RoboDK station: KR200-2_Roboforming_Escala_Laboratorio.rdk

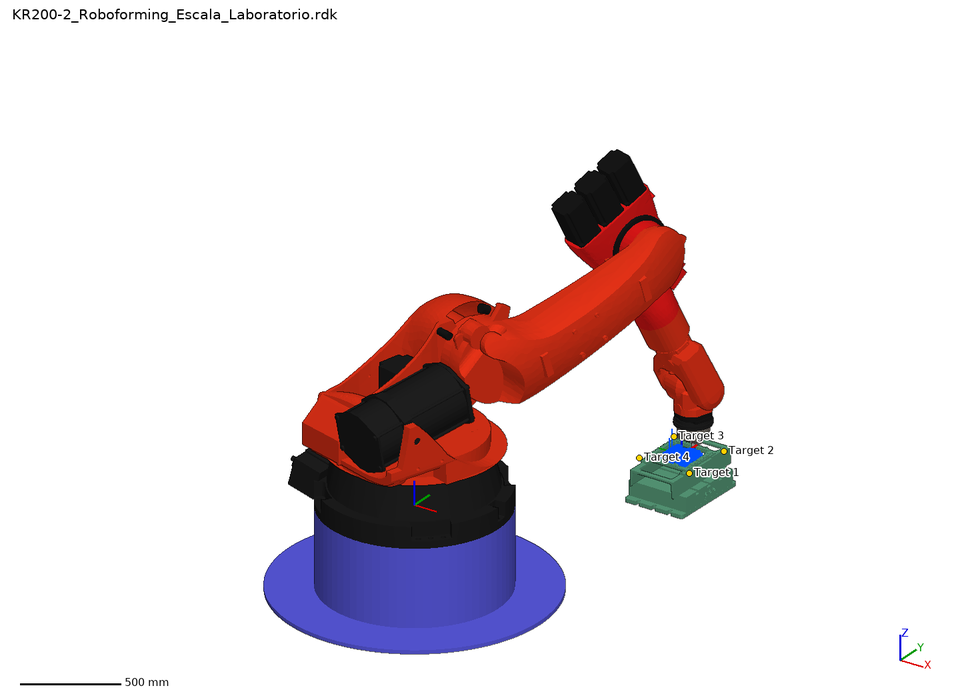
[picture v0: the station drawn from its stored meshes, robots at their saved joint values, targets as dots, program paths as lines]
Station KR200-2_Roboforming_Escala_Laboratorio (saved by RoboDK 5.8.0). Poses are relative to the parent item; angles as X-Y-Z fixed-axis rotations.
Station parameters (name, value as stored): IO_5, 1
  - frame KR200-2 comp Base at (0, 0, 458.56) mm
    - robot KR200-2 comp: 6 axes
        modified DH rows (alpha deg, a mm, theta deg, d mm): 0, 0, 0, 750; -90, 350, 0, 0; 0, 1050, -90, 0; -90, -45, 0, 1000; 90, 0, 0, 0; -90, 0, 180, 210
        joint limits [-185, -142, -120, -350, -120, -350] to [185, 0, 148, 350, 120, 350]; home [0, -90, 90, 0, 0, 0]; saved at [73.183, -16.623, 80.288, 0, 26.334, 73.183]
      - tool Kitagawa JN06T, TCP at (0, 0, 200) mm, size 164.9 x 165.3 x 101 mm, geometry from Kitagawa JN06T.STEP
      - tool herramienta_spif, TCP at (0, 0, 170) mm, size 17.5 x 18 x 175 mm, geometry from herramienta_spif.STEP
      - tool SPIF_TOOL, TCP at (0, 0, 170) mm, size 59.8 x 60 x 80 mm, geometry from SPIF_TOOL.stl
    - frame Machining at (474.42, 1634.58, -244.56) mm, rotated rx 0 ry 0 rz 90 deg
      - object myPart at (0, 0, 0) mm, size 300 x 300 x 40 mm, geometry from myPart.STP
        - object myToolpath_topToolTipPnts at (0, 0, 0) mm
      - target Target 1 (Cartesian target) at (-150, -150, 0) mm, rotated rx 179.98 ry -0.02 rz -135 deg; joints [14.532, -78.087, 109.692, 0.007, 58.419, -30.472] of KR200-2 comp
      - target Target 2 (Cartesian target) at (150, -150, 0) mm, rotated rx 179.98 ry -0.02 rz -135 deg; joints [11.975, -64.118, 90.175, 0.006, 63.968, -33.028] of KR200-2 comp
      - target Target 3 (Cartesian target) at (150, 150, 0) mm, rotated rx 179.98 ry -0.02 rz -135 deg; joints [21.499, -59.92, 83.648, 0.01, 66.295, -23.505] of KR200-2 comp
      - target Target 4 (Cartesian target) at (-150, 150, 0) mm, rotated rx 179.98 ry -0.02 rz -135 deg; joints [25.706, -73.09, 103.133, 0.013, 59.98, -19.3] of KR200-2 comp
  - machining project Machining1 settings: F:/SPIF.ptp | rotZ(0) | rotX(0)*rotY(0)
  - program Machining1 (10854 instructions, listed below)
  - object dispositivo sin pieza at (474.42, 1634.58, 214) mm, rotated rx 0 ry 0 rz 90 deg, size 500 x 358.5 x 227 mm, geometry from dispositivo sin pieza.STEP
  - object Base at (0, 0, 0) mm, size 1499.1 x 1499.1 x 458.6 mm, geometry from Base.IGS
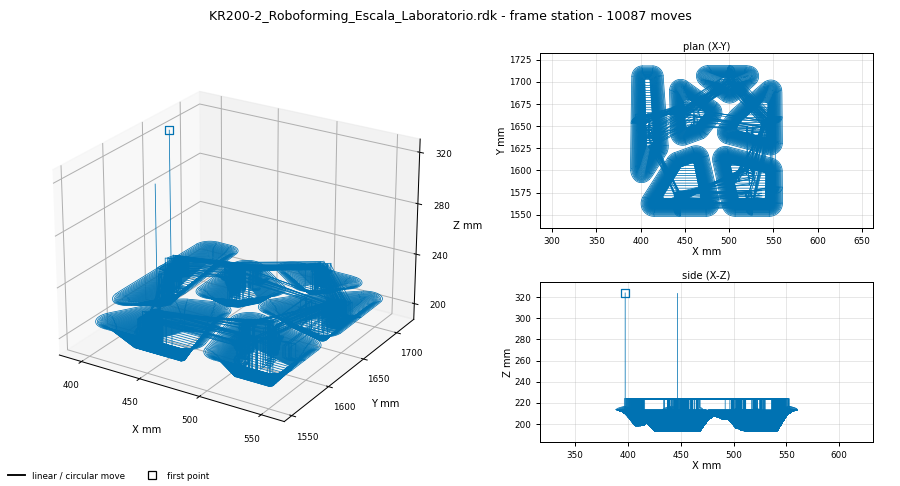
[picture p0: tool path of KR200-2_Roboforming_Escala_Laboratorio.rdk in frame station, 10087 of 10087 moves have a stored position in this frame; points joined in program order, loops and branches not executed]

--- program Machining1 (robot KR200-2 comp) ---
  Suave(1)
  Llamar SetTool(1)
  Llamar M_RunCode(6)
  Llamar SetRPM(0.0)
  Llamar M_RunCode(3)
  Establecer velocidad (1000.0 mm/s)
  Est. Ref.: Machining
  Est. herr: SPIF_TOOL
  Mostrar SPIF_TOOL
  MoveJ 1 to (25.11, 76.92, 110) mm, rotated rx 180 ry 0 rz 90 deg; joints [76.531, -23.354, 87.682, 0, 25.671, 76.531]
  MoveL 2 to (25.11, 76.92, 110) mm, rotated rx 180 ry 0 rz 90 deg; joints [76.531, -23.354, 87.682, 0, 25.671, 76.531]
  MoveL 3 to (25.11, 76.92, 10) mm, rotated rx -180 ry 0 rz 90 deg; joints [76.531, -18.294, 84.658, 0, 23.636, 76.531]
  MoveL 4 to (25.11, 76.92, 10) mm, rotated rx -180 ry 0 rz 90 deg; joints [76.531, -18.294, 84.658, 0, 23.636, 76.531]
  MoveL 5 to (25.11, 76.92, 10) mm, rotated rx -180 ry 0 rz 90 deg; joints [76.531, -18.294, 84.658, 0, 23.636, 76.531]
  MoveL 6 to (25.11, 76.92, 3) mm, rotated rx 180 ry 0 rz 90 deg; joints [76.531, -17.937, 84.426, 0, 23.511, 76.531]
  Establecer velocidad (66.7 mm/s)
  MoveL 7 to (25.32, 78.42, 2.59) mm, rotated rx 180 ry 0 rz 90 deg; joints [76.582, -17.919, 84.424, 0, 23.496, 76.582]
  MoveL 8 to (25.15, 79.93, 2.19) mm, rotated rx -180 ry 0 rz 90 deg; joints [76.63, -17.909, 84.448, 0, 23.461, 76.63]
  MoveL 9 to (24.66, 81.37, 1.78) mm, rotated rx -180 ry 0 rz 90 deg; joints [76.673, -17.904, 84.494, 0, 23.409, 76.673]
  MoveL 10 to (23.86, 82.66, 1.37) mm, rotated rx 180 ry 0 rz 90 deg; joints [76.709, -17.904, 84.56, 0, 23.344, 76.709]
  MoveL 11 to (22.79, 83.75, 0.97) mm, rotated rx 180 ry 0 rz 90 deg; joints [76.736, -17.908, 84.641, 0, 23.266, 76.736]
  MoveL 12 to (21.51, 84.57, 0.56) mm, rotated rx -180 ry 0 rz 90 deg; joints [76.753, -17.915, 84.734, 0, 23.181, 76.753]
  MoveL 13 to (20.09, 85.08, 0.16) mm, rotated rx 180 ry 0 rz 90 deg; joints [76.759, -17.923, 84.831, 0, 23.092, 76.759]
  MoveL 14 to (18.58, 85.24, -0.25) mm, rotated rx -180 ry 0 rz 90 deg; joints [76.753, -17.931, 84.928, 0, 23.002, 76.753]
  MoveL 15 to (-29.85, 85.86, -0.25) mm, rotated rx -180 ry 0 rz 90 deg; joints [76.389, -18.776, 88.341, 0, 20.435, 76.389]
  MoveL 16 to (-34.65, 85.65, -0.25) mm, rotated rx -180 ry 0 rz 90 deg; joints [76.342, -18.853, 88.668, 0, 20.185, 76.342]
  MoveC 17 to (-41.94, 83.49, -0.25) mm, rotated rx -180 ry 0 rz 90 deg; joints [76.209, -18.961, 89.132, 0, 19.829, 76.209] to (-47.38, 78.18, -0.25) mm, rotated rx -180 ry 0 rz 90 deg; joints [75.983, -19.025, 89.413, 0, 19.612, 75.983]
  MoveC 18 to (-48.12, 71.04, -0.25) mm, rotated rx 180 ry 0 rz 90 deg; joints [75.734, -19.009, 89.34, 0, 19.668, 75.734] to (-44.7, 64.73, -0.25) mm, rotated rx 180 ry 0 rz 90 deg; joints [75.55, -18.93, 88.997, 0, 19.932, 75.55]
  MoveL 19 to (-43.12, 63.19, -0.25) mm, rotated rx 180 ry 0 rz 90 deg; joints [75.512, -18.898, 88.862, 0, 20.036, 75.512]
  MoveL 20 to (-40.5, 61.12, -0.25) mm, rotated rx 180 ry 0 rz 90 deg; joints [75.465, -18.848, 88.647, 0, 20.201, 75.465]
  MoveL 21 to (-15.64, 45.37, -0.25) mm, rotated rx 180 ry 0 rz 90 deg; joints [75.157, -18.366, 86.643, 0, 21.723, 75.157]
  MoveL 22 to (-14.69, 44.91, -0.25) mm, rotated rx -180 ry 0 rz 90 deg; joints [75.15, -18.347, 86.568, 0, 21.779, 75.15]
  MoveC 23 to (-10.63, 43.57, -0.25) mm, rotated rx -180 ry 0 rz 90 deg; joints [75.141, -18.27, 86.259, 0, 22.011, 75.141] to (-6.36, 43.32, -0.25) mm, rotated rx 180 ry 0 rz 90 deg; joints [75.17, -18.193, 85.955, 0, 22.239, 75.17]
  MoveL 24 to (58.28, 48.02, -0.25) mm, rotated rx -180 ry 0 rz 90 deg; joints [75.862, -16.971, 81.374, 0, 25.597, 75.862]
  MoveL 25 to (72.44, 48.99, -0.25) mm, rotated rx -180 ry 0 rz 90 deg; joints [76.006, -16.677, 80.335, 0, 26.342, 76.006]
  MoveC 26 to (80.2, 52.59, -0.25) mm, rotated rx -180 ry 0 rz 90 deg; joints [76.18, -16.528, 79.817, 0, 26.711, 76.18] to (83.56, 60.47, -0.25) mm, rotated rx 180 ry 0 rz 90 deg; joints [76.454, -16.496, 79.708, 0, 26.788, 76.454]
  MoveL 27 to (83.58, 61.12, -0.25) mm, rotated rx -180 ry 0 rz 90 deg; joints [76.475, -16.499, 79.718, 0, 26.781, 76.475]
  MoveL 28 to (83.58, 72.42, -0.25) mm, rotated rx 180 ry 0 rz 90 deg; joints [76.831, -16.558, 79.921, 0, 26.637, 76.831]
  MoveC 29 to (80.15, 80.83, -0.25) mm, rotated rx 180 ry 0 rz 90 deg; joints [77.073, -16.675, 80.328, 0, 26.347, 77.073] to (71.81, 84.44, -0.25) mm, rotated rx 180 ry 0 rz 90 deg; joints [77.127, -16.871, 81.017, 0, 25.854, 77.127]
  MoveL 30 to (54.49, 84.79, -0.25) mm, rotated rx -180 ry 0 rz 90 deg; joints [77.01, -17.231, 82.31, 0, 24.921, 77.01]
  MoveL 31 to (18.58, 85.24, -0.25) mm, rotated rx -180 ry 0 rz 90 deg; joints [76.753, -17.931, 84.928, 0, 23.002, 76.753]
  MoveL 32 to (18.48, 77.69, -0.25) mm, rotated rx -180 ry 0 rz 90 deg; joints [76.505, -17.899, 84.807, 0, 23.093, 76.505]
  MoveL 33 to (18.48, 77.69, 2.75) mm, rotated rx -180 ry 0 rz 90 deg; joints [76.505, -18.053, 84.907, 0, 23.146, 76.505]
  Establecer velocidad (1000.0 mm/s)
  MoveL 34 to (18.48, 77.69, 10) mm, rotated rx 180 ry 0 rz 90 deg; joints [76.505, -18.423, 85.148, 0, 23.276, 76.505]
  Establecer velocidad (66.7 mm/s)
  MoveL 35 to (38.08, 33.07, 10) mm, rotated rx 180 ry 0 rz 90 deg; joints [75.219, -17.824, 82.918, 0, 24.906, 75.219]
  MoveL 36 to (38.08, 33.07, 3) mm, rotated rx -180 ry 0 rz 90 deg; joints [75.219, -17.469, 82.685, 0, 24.784, 75.219]
  MoveL 37 to (38.23, 34.58, 2.59) mm, rotated rx 180 ry 0 rz 90 deg; joints [75.269, -17.454, 82.69, 0, 24.763, 75.269]
  MoveL 38 to (38, 36.09, 2.19) mm, rotated rx 180 ry 0 rz 90 deg; joints [75.315, -17.445, 82.722, 0, 24.723, 75.315]
  MoveL 39 to (37.45, 37.5, 1.78) mm, rotated rx -180 ry 0 rz 90 deg; joints [75.356, -17.443, 82.776, 0, 24.668, 75.356]
  MoveL 40 to (36.6, 38.76, 1.37) mm, rotated rx 180 ry 0 rz 90 deg; joints [75.389, -17.446, 82.848, 0, 24.598, 75.389]
  MoveL 41 to (35.49, 39.8, 0.97) mm, rotated rx 180 ry 0 rz 90 deg; joints [75.413, -17.453, 82.935, 0, 24.518, 75.413]
  MoveL 42 to (34.18, 40.57, 0.56) mm, rotated rx -180 ry 0 rz 90 deg; joints [75.427, -17.462, 83.031, 0, 24.431, 75.427]
  MoveL 43 to (32.74, 41.03, 0.16) mm, rotated rx -180 ry 0 rz 90 deg; joints [75.429, -17.472, 83.131, 0, 24.341, 75.429]
  MoveL 44 to (31.22, 41.13, -0.25) mm, rotated rx -180 ry 0 rz 90 deg; joints [75.42, -17.482, 83.229, 0, 24.252, 75.42]
  MoveL 45 to (7.11, 40.47, -0.25) mm, rotated rx -180 ry 0 rz 90 deg; joints [75.193, -17.936, 84.949, 0, 22.987, 75.193]
  MoveL 46 to (5.6, 40.3, -0.25) mm, rotated rx 180 ry 0 rz 90 deg; joints [75.175, -17.963, 85.052, 0, 22.911, 75.175]
  MoveC 47 to (-4.04, 34.34, -0.25) mm, rotated rx 180 ry 0 rz 90 deg; joints [74.896, -18.109, 85.622, 0, 22.487, 74.896] to (-5.53, 23.11, -0.25) mm, rotated rx -180 ry 0 rz 90 deg; joints [74.515, -18.081, 85.511, 0, 22.57, 74.515]
  MoveL 48 to (-4.96, 21.32, -0.25) mm, rotated rx -180 ry 0 rz 90 deg; joints [74.462, -18.062, 85.436, 0, 22.626, 74.462]
  MoveL 49 to (0.91, 5.21, -0.25) mm, rotated rx -180 ry 0 rz 90 deg; joints [73.992, -17.871, 84.699, 0, 23.172, 73.992]
  MoveL 50 to (1.74, 3.32, -0.25) mm, rotated rx 180 ry 0 rz 90 deg; joints [73.939, -17.846, 84.602, 0, 23.244, 73.939]
  MoveC 51 to (3.62, 0.75, -0.25) mm, rotated rx 180 ry 0 rz 90 deg; joints [73.873, -17.797, 84.416, 0, 23.382, 73.873] to (5.93, -1.42, -0.25) mm, rotated rx 180 ry 0 rz 90 deg; joints [73.825, -17.742, 84.206, 0, 23.536, 73.825]
  MoveL 52 to (22.27, -14.11, -0.25) mm, rotated rx -180 ry 0 rz 90 deg; joints [73.572, -17.357, 82.768, 0, 24.589, 73.572]
  MoveL 53 to (23.38, -14.89, -0.25) mm, rotated rx 180 ry 0 rz 90 deg; joints [73.557, -17.33, 82.671, 0, 24.659, 73.557]
  MoveC 54 to (33.35, -17.16, -0.25) mm, rotated rx -180 ry 0 rz 90 deg; joints [73.579, -17.117, 81.898, 0, 25.219, 73.579] to (42.02, -11.74, -0.25) mm, rotated rx -180 ry 0 rz 90 deg; joints [73.83, -16.973, 81.379, 0, 25.593, 73.83]
  MoveL 55 to (65.02, 20.37, -0.25) mm, rotated rx 180 ry 0 rz 90 deg; joints [75.043, -16.677, 80.337, 0, 26.34, 75.043]
  MoveL 56 to (66.39, 22.51, -0.25) mm, rotated rx 180 ry 0 rz 90 deg; joints [75.122, -16.66, 80.277, 0, 26.383, 75.122]
  MoveC 57 to (67.04, 34.78, -0.25) mm, rotated rx 180 ry 0 rz 90 deg; joints [75.514, -16.715, 80.469, 0, 26.246, 75.514] to (56.85, 41.63, -0.25) mm, rotated rx 180 ry 0 rz 90 deg; joints [75.648, -16.967, 81.36, 0, 25.607, 75.648]
  MoveL 58 to (55.44, 41.74, -0.25) mm, rotated rx 180 ry 0 rz 90 deg; joints [75.639, -16.997, 81.466, 0, 25.531, 75.639]
  MoveL 59 to (54.49, 41.77, -0.25) mm, rotated rx -180 ry 0 rz 90 deg; joints [75.633, -17.017, 81.537, 0, 25.48, 75.633]
  MoveL 60 to (31.22, 41.13, -0.25) mm, rotated rx -180 ry 0 rz 90 deg; joints [75.42, -17.482, 83.229, 0, 24.252, 75.42]
  MoveL 61 to (31.43, 33.58, -0.25) mm, rotated rx -180 ry 0 rz 90 deg; joints [75.179, -17.439, 83.071, 0, 24.368, 75.179]
  MoveL 62 to (31.43, 33.58, 2.75) mm, rotated rx -180 ry 0 rz 90 deg; joints [75.179, -17.591, 83.171, 0, 24.42, 75.179]
  Establecer velocidad (1000.0 mm/s)
  MoveL 63 to (31.43, 33.58, 10) mm, rotated rx 180 ry 0 rz 90 deg; joints [75.179, -17.959, 83.412, 0, 24.547, 75.179]
  Establecer velocidad (66.7 mm/s)
  MoveL 64 to (75.76, -31.94, 10) mm, rotated rx 180 ry 0 rz 90 deg; joints [73.508, -16.63, 78.763, 0, 27.867, 73.508]
  MoveL 65 to (75.76, -31.94, 3) mm, rotated rx -180 ry 0 rz 90 deg; joints [73.508, -16.281, 78.529, 0, 27.752, 73.508]
  MoveL 66 to (77.26, -32.13, 2.59) mm, rotated rx 180 ry 0 rz 90 deg; joints [73.516, -16.225, 78.396, 0, 27.829, 73.516]
  MoveL 67 to (78.77, -31.95, 2.19) mm, rotated rx 180 ry 0 rz 90 deg; joints [73.535, -16.172, 78.272, 0, 27.9, 73.535]
  MoveL 68 to (80.2, -31.43, 1.78) mm, rotated rx 180 ry 0 rz 90 deg; joints [73.564, -16.123, 78.161, 0, 27.962, 73.564]
  MoveL 69 to (81.48, -30.62, 1.37) mm, rotated rx -180 ry 0 rz 90 deg; joints [73.601, -16.079, 78.068, 0, 28.011, 73.601]
  MoveL 70 to (82.56, -29.54, 0.97) mm, rotated rx 180 ry 0 rz 90 deg; joints [73.644, -16.041, 77.997, 0, 28.045, 73.644]
  MoveL 71 to (83.36, -28.25, 0.56) mm, rotated rx -180 ry 0 rz 90 deg; joints [73.69, -16.011, 77.95, 0, 28.061, 73.69]
  MoveL 72 to (83.86, -26.81, 0.16) mm, rotated rx -180 ry 0 rz 90 deg; joints [73.739, -15.989, 77.93, 0, 28.059, 73.739]
  MoveL 73 to (84, -25.3, -0.25) mm, rotated rx -180 ry 0 rz 90 deg; joints [73.787, -15.976, 77.94, 0, 28.036, 73.787]
  MoveL 74 to (84, -4.26, -0.25) mm, rotated rx -180 ry 0 rz 90 deg; joints [74.436, -16.112, 78.397, 0, 27.715, 74.436]
  MoveL 75 to (83.9, -1.36, -0.25) mm, rotated rx 180 ry 0 rz 90 deg; joints [74.525, -16.132, 78.466, 0, 27.667, 74.525]
  MoveC 76 to (81.73, 5.7, -0.25) mm, rotated rx -180 ry 0 rz 90 deg; joints [74.725, -16.225, 78.779, 0, 27.446, 74.725] to (76.29, 10.7, -0.25) mm, rotated rx -180 ry 0 rz 90 deg; joints [74.835, -16.376, 79.294, 0, 27.082, 74.835]
  MoveC 77 to (69.05, 10.89, -0.25) mm, rotated rx 180 ry 0 rz 90 deg; joints [74.779, -16.535, 79.844, 0, 26.692, 74.779] to (62.94, 7.01, -0.25) mm, rotated rx -180 ry 0 rz 90 deg; joints [74.605, -16.644, 80.222, 0, 26.423, 74.605]
  MoveL 78 to (60.58, 4.26, -0.25) mm, rotated rx 180 ry 0 rz 90 deg; joints [74.499, -16.679, 80.341, 0, 26.337, 74.499]
  MoveL 79 to (44.7, -17.53, -0.25) mm, rotated rx -180 ry 0 rz 90 deg; joints [73.672, -16.882, 81.058, 0, 25.824, 73.672]
  MoveL 80 to (43.76, -18.94, -0.25) mm, rotated rx 180 ry 0 rz 90 deg; joints [73.619, -16.893, 81.097, 0, 25.797, 73.619]
  MoveC 81 to (41.63, -26.99, -0.25) mm, rotated rx 180 ry 0 rz 90 deg; joints [73.346, -16.888, 81.078, 0, 25.81, 73.346] to (44.86, -34.66, -0.25) mm, rotated rx -180 ry 0 rz 90 deg; joints [73.137, -16.772, 80.669, 0, 26.103, 73.137]
  MoveL 82 to (62.52, -54.49, -0.25) mm, rotated rx -180 ry 0 rz 90 deg; joints [72.69, -16.261, 78.901, 0, 27.36, 72.69]
  MoveL 83 to (63.6, -55.44, -0.25) mm, rotated rx -180 ry 0 rz 90 deg; joints [72.671, -16.23, 78.797, 0, 27.433, 72.671]
  MoveL 84 to (64.56, -56.24, -0.25) mm, rotated rx -180 ry 0 rz 90 deg; joints [72.656, -16.204, 78.707, 0, 27.497, 72.656]
  MoveC 85 to (75.98, -58.19, -0.25) mm, rotated rx -180 ry 0 rz 90 deg; joints [72.705, -15.933, 77.796, 0, 28.137, 72.705] to (83.3, -49.2, -0.25) mm, rotated rx 180 ry 0 rz 90 deg; joints [73.048, -15.829, 77.449, 0, 28.38, 73.048]
  MoveL 86 to (83.95, -45.01, -0.25) mm, rotated rx -180 ry 0 rz 90 deg; joints [73.182, -15.843, 77.496, 0, 28.346, 73.182]
  MoveL 87 to (84, -44.07, -0.25) mm, rotated rx -180 ry 0 rz 90 deg; joints [73.212, -15.848, 77.515, 0, 28.334, 73.212]
  MoveL 88 to (84, -25.3, -0.25) mm, rotated rx -180 ry 0 rz 90 deg; joints [73.787, -15.976, 77.94, 0, 28.036, 73.787]
  MoveL 89 to (76.45, -25.3, -0.25) mm, rotated rx 180 ry 0 rz 90 deg; joints [73.719, -16.147, 78.514, 0, 27.632, 73.719]
  MoveL 90 to (76.45, -25.3, 2.75) mm, rotated rx 180 ry 0 rz 90 deg; joints [73.719, -16.297, 78.616, 0, 27.681, 73.719]
  Establecer velocidad (1000.0 mm/s)
  MoveL 91 to (76.45, -25.3, 10) mm, rotated rx -180 ry 0 rz 90 deg; joints [73.719, -16.659, 78.859, 0, 27.8, 73.719]
  Establecer velocidad (66.7 mm/s)
  MoveL 92 to (19.29, -77.28, 10) mm, rotated rx -180 ry 0 rz 90 deg; joints [71.552, -17.537, 81.89, 0, 25.648, 71.552]
  MoveL 93 to (19.29, -77.28, 3) mm, rotated rx 180 ry 0 rz 90 deg; joints [71.552, -17.184, 81.656, 0, 25.527, 71.552]
  MoveL 94 to (19.12, -78.79, 2.59) mm, rotated rx 180 ry 0 rz 90 deg; joints [71.503, -17.157, 81.619, 0, 25.538, 71.503]
  MoveL 95 to (19.32, -80.3, 2.19) mm, rotated rx 180 ry 0 rz 90 deg; joints [71.458, -17.122, 81.554, 0, 25.568, 71.458]
  MoveL 96 to (19.85, -81.72, 1.78) mm, rotated rx 180 ry 0 rz 90 deg; joints [71.42, -17.081, 81.468, 0, 25.613, 71.42]
  MoveL 97 to (20.67, -83, 1.37) mm, rotated rx 180 ry 0 rz 90 deg; joints [71.389, -17.035, 81.363, 0, 25.672, 71.389]
  MoveL 98 to (21.76, -84.06, 0.97) mm, rotated rx 180 ry 0 rz 90 deg; joints [71.367, -16.985, 81.244, 0, 25.74, 71.367]
  MoveL 99 to (23.06, -84.85, 0.56) mm, rotated rx 180 ry 0 rz 90 deg; joints [71.356, -16.932, 81.117, 0, 25.815, 71.356]
  MoveL 100 to (24.5, -85.34, 0.16) mm, rotated rx 180 ry 0 rz 90 deg; joints [71.356, -16.879, 80.987, 0, 25.892, 71.356]
  MoveL 101 to (26.01, -85.46, -0.25) mm, rotated rx -180 ry 0 rz 90 deg; joints [71.368, -16.826, 80.86, 0, 25.966, 71.368]
  MoveL 102 to (53.54, -85.2, -0.25) mm, rotated rx 180 ry 0 rz 90 deg; joints [71.659, -16.241, 78.834, 0, 27.407, 71.659]
  MoveL 103 to (56.28, -84.98, -0.25) mm, rotated rx -180 ry 0 rz 90 deg; joints [71.694, -16.182, 78.634, 0, 27.548, 71.694]
  MoveC 104 to (66.45, -77.93, -0.25) mm, rotated rx 180 ry 0 rz 90 deg; joints [72.011, -16.007, 78.043, 0, 27.964, 72.011] to (65.33, -65.6, -0.25) mm, rotated rx 180 ry 0 rz 90 deg; joints [72.376, -16.121, 78.426, 0, 27.694, 72.376]
  MoveL 105 to (63.5, -63.02, -0.25) mm, rotated rx 180 ry 0 rz 90 deg; joints [72.438, -16.18, 78.626, 0, 27.554, 72.438]
  MoveL 106 to (34.59, -29.56, -0.25) mm, rotated rx 180 ry 0 rz 90 deg; joints [73.199, -17.017, 81.538, 0, 25.48, 73.199]
  MoveL 107 to (33.64, -28.5, -0.25) mm, rotated rx 180 ry 0 rz 90 deg; joints [73.223, -17.043, 81.63, 0, 25.413, 73.223]
  MoveL 108 to (33.08, -27.96, -0.25) mm, rotated rx -180 ry 0 rz 90 deg; joints [73.235, -17.058, 81.683, 0, 25.374, 73.235]
  MoveL 109 to (17.53, -15.48, -0.25) mm, rotated rx 180 ry 0 rz 90 deg; joints [73.483, -17.441, 83.081, 0, 24.361, 73.483]
  MoveL 110 to (15.92, -14.42, -0.25) mm, rotated rx 180 ry 0 rz 90 deg; joints [73.502, -17.479, 83.219, 0, 24.26, 73.502]
  MoveC 111 to (3.85, -13.12, -0.25) mm, rotated rx 180 ry 0 rz 90 deg; joints [73.429, -17.717, 84.109, 0, 23.607, 73.429] to (-4.25, -22.15, -0.25) mm, rotated rx -180 ry 0 rz 90 deg; joints [73.06, -17.817, 84.492, 0, 23.326, 73.06]
  MoveL 112 to (-16.58, -68.7, -0.25) mm, rotated rx 180 ry 0 rz 90 deg; joints [71.444, -17.769, 84.31, 0, 23.46, 71.444]
  MoveC 113 to (-14.48, -80.13, -0.25) mm, rotated rx -180 ry 0 rz 90 deg; joints [71.104, -17.659, 83.89, 0, 23.768, 71.104] to (-4.26, -85.66, -0.25) mm, rotated rx -180 ry 0 rz 90 deg; joints [71.04, -17.429, 83.034, 0, 24.395, 71.04]
  MoveL 114 to (-2.37, -85.73, -0.25) mm, rotated rx -180 ry 0 rz 90 deg; joints [71.059, -17.392, 82.897, 0, 24.494, 71.059]
  MoveL 115 to (26.01, -85.46, -0.25) mm, rotated rx -180 ry 0 rz 90 deg; joints [71.368, -16.826, 80.86, 0, 25.966, 71.368]
  MoveL 116 to (25.94, -77.91, -0.25) mm, rotated rx -180 ry 0 rz 90 deg; joints [71.602, -16.88, 81.049, 0, 25.831, 71.602]
  MoveL 117 to (25.94, -77.91, 2.75) mm, rotated rx -180 ry 0 rz 90 deg; joints [71.602, -17.031, 81.15, 0, 25.881, 71.602]
  Establecer velocidad (1000.0 mm/s)
  MoveL 118 to (25.94, -77.91, 10) mm, rotated rx 180 ry 0 rz 90 deg; joints [71.602, -17.396, 81.392, 0, 26.004, 71.602]
  Establecer velocidad (66.7 mm/s)
  MoveL 119 to (-60.09, -77.51, 10) mm, rotated rx -180 ry 0 rz 90 deg; joints [70.682, -19.008, 87.445, 0, 21.563, 70.682]
  MoveL 120 to (-60.09, -77.51, 3) mm, rotated rx 180 ry 0 rz 90 deg; joints [70.682, -18.647, 87.213, 0, 21.434, 70.682]
  MoveL 121 to (-60.27, -79.01, 2.59) mm, rotated rx 180 ry 0 rz 90 deg; joints [70.631, -18.62, 87.175, 0, 21.445, 70.631]
  MoveL 122 to (-60.07, -80.52, 2.19) mm, rotated rx -180 ry 0 rz 90 deg; joints [70.585, -18.587, 87.113, 0, 21.474, 70.585]
  MoveL 123 to (-59.55, -81.95, 1.78) mm, rotated rx -180 ry 0 rz 90 deg; joints [70.545, -18.549, 87.029, 0, 21.52, 70.545]
  MoveL 124 to (-58.72, -83.22, 1.37) mm, rotated rx -180 ry 0 rz 90 deg; joints [70.513, -18.507, 86.929, 0, 21.577, 70.513]
  MoveL 125 to (-57.64, -84.28, 0.97) mm, rotated rx -180 ry 0 rz 90 deg; joints [70.491, -18.461, 86.816, 0, 21.645, 70.491]
  MoveL 126 to (-56.34, -85.08, 0.56) mm, rotated rx 180 ry 0 rz 90 deg; joints [70.48, -18.414, 86.695, 0, 21.718, 70.48]
  MoveL 127 to (-54.9, -85.57, 0.16) mm, rotated rx 180 ry 0 rz 90 deg; joints [70.481, -18.366, 86.572, 0, 21.794, 70.481]
  MoveL 128 to (-53.39, -85.69, -0.25) mm, rotated rx -180 ry 0 rz 90 deg; joints [70.494, -18.318, 86.452, 0, 21.866, 70.494]
  MoveL 129 to (-35.3, -85.56, -0.25) mm, rotated rx -180 ry 0 rz 90 deg; joints [70.703, -18.004, 85.212, 0, 22.792, 70.703]
  MoveC 130 to (-26.15, -82.38, -0.25) mm, rotated rx 180 ry 0 rz 90 deg; joints [70.905, -17.859, 84.654, 0, 23.206, 70.905] to (-20.83, -74.28, -0.25) mm, rotated rx -180 ry 0 rz 90 deg; joints [71.221, -17.813, 84.476, 0, 23.337, 71.221]
  MoveL 131 to (-8.05, -25.1, -0.25) mm, rotated rx -180 ry 0 rz 90 deg; joints [72.928, -17.871, 84.696, 0, 23.174, 72.928]
  MoveC 132 to (-11.52, -11.33, -0.25) mm, rotated rx -180 ry 0 rz 90 deg; joints [73.339, -18.01, 85.234, 0, 22.776, 73.339] to (-25.11, -7.26, -0.25) mm, rotated rx -180 ry 0 rz 90 deg; joints [73.339, -18.272, 86.269, 0, 22.004, 73.339]
  MoveL 133 to (-74.68, -17.81, -0.25) mm, rotated rx 180 ry 0 rz 90 deg; joints [72.487, -19.028, 89.426, 0, 19.602, 72.487]
  MoveC 134 to (-83.14, -22.99, -0.25) mm, rotated rx 180 ry 0 rz 90 deg; joints [72.223, -19.131, 89.88, 0, 19.25, 72.223] to (-86.46, -32.35, -0.25) mm, rotated rx 180 ry 0 rz 90 deg; joints [71.874, -19.135, 89.899, 0, 19.236, 71.874]
  MoveL 135 to (-86.48, -70.94, -0.25) mm, rotated rx -180 ry 0 rz 90 deg; joints [70.594, -18.937, 89.03, 0, 19.907, 70.594]
  MoveC 136 to (-82.08, -81.51, -0.25) mm, rotated rx 180 ry 0 rz 90 deg; joints [70.298, -18.811, 88.488, 0, 20.323, 70.298] to (-71.48, -85.83, -0.25) mm, rotated rx -180 ry 0 rz 90 deg; joints [70.281, -18.618, 87.674, 0, 20.943, 70.281]
  MoveL 137 to (-53.39, -85.69, -0.25) mm, rotated rx -180 ry 0 rz 90 deg; joints [70.494, -18.318, 86.452, 0, 21.866, 70.494]
  MoveL 138 to (-53.45, -78.15, -0.25) mm, rotated rx 180 ry 0 rz 90 deg; joints [70.737, -18.364, 86.637, 0, 21.727, 70.737]
  MoveL 139 to (-53.45, -78.15, 2.75) mm, rotated rx 180 ry 0 rz 90 deg; joints [70.737, -18.519, 86.738, 0, 21.781, 70.737]
  Establecer velocidad (1000.0 mm/s)
  MoveL 140 to (-53.45, -78.15, 10) mm, rotated rx -180 ry 0 rz 90 deg; joints [70.737, -18.892, 86.978, 0, 21.914, 70.737]
  Establecer velocidad (66.7 mm/s)
  MoveL 141 to (-78.23, 36.45, 10) mm, rotated rx 180 ry 0 rz 90 deg; joints [74.283, -19.86, 91.085, 0, 18.775, 74.283]
  MoveL 142 to (-78.23, 36.45, 3) mm, rotated rx -180 ry 0 rz 90 deg; joints [74.283, -19.493, 90.853, 0, 18.64, 74.283]
  MoveL 143 to (-79.74, 36.64, 2.59) mm, rotated rx -180 ry 0 rz 90 deg; joints [74.275, -19.494, 90.943, 0, 18.551, 74.275]
  MoveL 144 to (-81.24, 36.45, 2.19) mm, rotated rx 180 ry 0 rz 90 deg; joints [74.254, -19.493, 91.026, 0, 18.468, 74.254]
  MoveL 145 to (-82.67, 35.94, 1.78) mm, rotated rx -180 ry 0 rz 90 deg; joints [74.223, -19.491, 91.098, 0, 18.393, 74.223]
  MoveL 146 to (-83.96, 35.13, 1.37) mm, rotated rx 180 ry 0 rz 90 deg; joints [74.182, -19.484, 91.154, 0, 18.33, 74.182]
  MoveL 147 to (-85.03, 34.05, 0.97) mm, rotated rx -180 ry 0 rz 90 deg; joints [74.135, -19.474, 91.191, 0, 18.283, 74.135]
  MoveL 148 to (-85.83, 32.76, 0.56) mm, rotated rx 180 ry 0 rz 90 deg; joints [74.083, -19.459, 91.206, 0, 18.252, 74.083]
  MoveL 149 to (-86.33, 31.32, 0.16) mm, rotated rx -180 ry 0 rz 90 deg; joints [74.029, -19.439, 91.199, 0, 18.24, 74.029]
  MoveL 150 to (-86.47, 29.81, -0.25) mm, rotated rx 180 ry 0 rz 90 deg; joints [73.976, -19.413, 91.166, 0, 18.247, 73.976]
  MoveL 151 to (-86.47, 0.4, -0.25) mm, rotated rx -180 ry 0 rz 90 deg; joints [72.976, -19.288, 90.588, 0, 18.7, 72.976]
  MoveC 152 to (-80.93, -11.12, -0.25) mm, rotated rx -180 ry 0 rz 90 deg; joints [72.645, -19.154, 89.983, 0, 19.171, 72.645] to (-68.46, -13.96, -0.25) mm, rotated rx 180 ry 0 rz 90 deg; joints [72.68, -18.951, 89.09, 0, 19.861, 72.68]
  MoveL 153 to (-58.28, -11.64, -0.25) mm, rotated rx -180 ry 0 rz 90 deg; joints [72.863, -18.803, 88.452, 0, 20.35, 72.863]
  MoveL 154 to (-19.43, -2.7, -0.25) mm, rotated rx -180 ry 0 rz 90 deg; joints [73.543, -18.197, 85.967, 0, 22.229, 73.543]
  MoveL 155 to (-17.83, -2.31, -0.25) mm, rotated rx 180 ry 0 rz 90 deg; joints [73.571, -18.17, 85.864, 0, 22.307, 73.571]
  MoveC 156 to (-8.42, 4.98, -0.25) mm, rotated rx 180 ry 0 rz 90 deg; joints [73.898, -18.04, 85.353, 0, 22.687, 73.898] to (-7.54, 16.85, -0.25) mm, rotated rx 180 ry 0 rz 90 deg; joints [74.292, -18.085, 85.529, 0, 22.556, 74.292]
  MoveL 157 to (-14.62, 36.55, -0.25) mm, rotated rx 180 ry 0 rz 90 deg; joints [74.875, -18.307, 86.407, 0, 21.9, 74.875]
  MoveC 158 to (-17.05, 40.7, -0.25) mm, rotated rx -180 ry 0 rz 90 deg; joints [74.99, -18.368, 86.654, 0, 21.714, 74.99] to (-20.65, 43.89, -0.25) mm, rotated rx -180 ry 0 rz 90 deg; joints [75.064, -18.445, 86.964, 0, 21.481, 75.064]
  MoveL 159 to (-63.02, 71.07, -0.25) mm, rotated rx 180 ry 0 rz 90 deg; joints [75.605, -19.235, 90.349, 0, 18.886, 75.605]
  MoveL 160 to (-64.91, 72.11, -0.25) mm, rotated rx 180 ry 0 rz 90 deg; joints [75.624, -19.267, 90.494, 0, 18.773, 75.624]
  MoveC 161 to (-79.41, 71.9, -0.25) mm, rotated rx -180 ry 0 rz 90 deg; joints [75.489, -19.476, 91.46, 0, 18.016, 75.489] to (-86.47, 59.23, -0.25) mm, rotated rx 180 ry 0 rz 90 deg; joints [74.987, -19.528, 91.706, 0, 17.822, 74.987]
  MoveL 162 to (-86.47, 29.81, -0.25) mm, rotated rx 180 ry 0 rz 90 deg; joints [73.976, -19.413, 91.166, 0, 18.247, 73.976]
  MoveL 163 to (-78.92, 29.81, -0.25) mm, rotated rx 180 ry 0 rz 90 deg; joints [74.05, -19.305, 90.664, 0, 18.64, 74.05]
  MoveL 164 to (-78.92, 29.81, 2.75) mm, rotated rx 180 ry 0 rz 90 deg; joints [74.05, -19.462, 90.765, 0, 18.697, 74.05]
  Establecer velocidad (1000.0 mm/s)
  MoveL 165 to (-78.92, 29.81, 10) mm, rotated rx -180 ry 0 rz 90 deg; joints [74.05, -19.843, 91.006, 0, 18.837, 74.05]
  Establecer velocidad (66.7 mm/s)
  MoveL 166 to (-77, 36.45, 10) mm, rotated rx -180 ry 0 rz 90 deg; joints [74.295, -19.842, 91.003, 0, 18.839, 74.295]
  MoveL 167 to (-77, 36.45, 2.75) mm, rotated rx 180 ry 0 rz 90 deg; joints [74.295, -19.461, 90.762, 0, 18.699, 74.295]
  MoveL 168 to (-78.5, 36.64, 2.34) mm, rotated rx 180 ry 0 rz 90 deg; joints [74.287, -19.463, 90.852, 0, 18.611, 74.287]
  MoveL 169 to (-80.01, 36.45, 1.94) mm, rotated rx -180 ry 0 rz 90 deg; joints [74.266, -19.463, 90.936, 0, 18.527, 74.266]
  MoveL 170 to (-81.44, 35.94, 1.53) mm, rotated rx 180 ry 0 rz 90 deg; joints [74.235, -19.46, 91.007, 0, 18.452, 74.235]
  MoveL 171 to (-82.72, 35.13, 1.13) mm, rotated rx 180 ry 0 rz 90 deg; joints [74.194, -19.454, 91.064, 0, 18.39, 74.194]
  MoveL 172 to (-83.79, 34.05, 0.72) mm, rotated rx 180 ry 0 rz 90 deg; joints [74.147, -19.443, 91.101, 0, 18.342, 74.147]
  MoveL 173 to (-84.6, 32.76, 0.31) mm, rotated rx -180 ry 0 rz 90 deg; joints [74.095, -19.428, 91.116, 0, 18.312, 74.095]
  MoveL 174 to (-85.1, 31.32, -0.09) mm, rotated rx -180 ry 0 rz 90 deg; joints [74.041, -19.408, 91.108, 0, 18.299, 74.041]
  MoveL 175 to (-85.23, 29.81, -0.5) mm, rotated rx 180 ry 0 rz 90 deg; joints [73.988, -19.382, 91.075, 0, 18.307, 73.988]
  MoveL 176 to (-85.24, 0.32, -0.5) mm, rotated rx -180 ry 0 rz 90 deg; joints [72.986, -19.256, 90.496, 0, 18.76, 72.986]
  MoveC 177 to (-80.7, -9.73, -0.5) mm, rotated rx 180 ry 0 rz 90 deg; joints [72.694, -19.144, 89.988, 0, 19.156, 72.694] to (-70.15, -12.95, -0.5) mm, rotated rx 180 ry 0 rz 90 deg; joints [72.697, -18.969, 89.216, 0, 19.753, 72.697]
  MoveL 178 to (-68.7, -12.76, -0.5) mm, rotated rx -180 ry 0 rz 90 deg; joints [72.718, -18.948, 89.123, 0, 19.824, 72.718]
  MoveL 179 to (-18.29, -1.16, -0.5) mm, rotated rx -180 ry 0 rz 90 deg; joints [73.604, -18.172, 85.911, 0, 22.261, 73.604]
  MoveC 180 to (-9.57, 5.44, -0.5) mm, rotated rx 180 ry 0 rz 90 deg; joints [73.902, -18.051, 85.435, 0, 22.616, 73.902] to (-8.7, 16.34, -0.5) mm, rotated rx 180 ry 0 rz 90 deg; joints [74.265, -18.091, 85.592, 0, 22.498, 74.265]
  MoveL 181 to (-15.6, 35.7, -0.5) mm, rotated rx 180 ry 0 rz 90 deg; joints [74.838, -18.307, 86.451, 0, 21.856, 74.838]
  MoveC 182 to (-17.85, 39.75, -0.5) mm, rotated rx 180 ry 0 rz 90 deg; joints [74.951, -18.365, 86.684, 0, 21.681, 74.951] to (-21.28, 42.85, -0.5) mm, rotated rx -180 ry 0 rz 90 deg; joints [75.024, -18.438, 86.981, 0, 21.457, 75.024]
  MoveL 183 to (-63.97, 70.21, -0.5) mm, rotated rx -180 ry 0 rz 90 deg; joints [75.568, -19.233, 90.389, 0, 18.843, 75.568]
  MoveL 184 to (-65.46, 71.03, -0.5) mm, rotated rx 180 ry 0 rz 90 deg; joints [75.582, -19.258, 90.504, 0, 18.754, 75.582]
  MoveC 185 to (-73.51, 72.61, -0.5) mm, rotated rx 180 ry 0 rz 90 deg; joints [75.566, -19.381, 91.07, 0, 18.311, 75.566] to (-81.02, 69.3, -0.5) mm, rotated rx 180 ry 0 rz 90 deg; joints [75.384, -19.476, 91.513, 0, 17.962, 75.384]
  MoveC 186 to (-84.14, 64.68, -0.5) mm, rotated rx -180 ry 0 rz 90 deg; joints [75.197, -19.502, 91.639, 0, 17.863, 75.197] to (-85.23, 59.23, -0.5) mm, rotated rx 180 ry 0 rz 90 deg; joints [74.998, -19.497, 91.616, 0, 17.882, 74.998]
  MoveL 187 to (-85.23, 29.81, -0.5) mm, rotated rx 180 ry 0 rz 90 deg; joints [73.988, -19.382, 91.075, 0, 18.307, 73.988]
  MoveL 188 to (-77.69, 29.81, -0.5) mm, rotated rx -180 ry 0 rz 90 deg; joints [74.062, -19.273, 90.574, 0, 18.7, 74.062]
  MoveL 189 to (-77.69, 29.81, 2.5) mm, rotated rx 180 ry 0 rz 90 deg; joints [74.062, -19.431, 90.674, 0, 18.757, 74.062]
  Establecer velocidad (1000.0 mm/s)
  MoveL 190 to (-77.69, 29.81, 10) mm, rotated rx 180 ry 0 rz 90 deg; joints [74.062, -19.824, 90.923, 0, 18.901, 74.062]
  Establecer velocidad (66.7 mm/s)
  MoveL 191 to (-77, -45.03, 10) mm, rotated rx -180 ry 0 rz 90 deg; joints [71.557, -19.462, 89.332, 0, 20.13, 71.557]
  MoveL 192 to (-77, -45.03, 2.75) mm, rotated rx 180 ry 0 rz 90 deg; joints [71.557, -19.084, 89.091, 0, 19.993, 71.557]
  MoveL 193 to (-78.51, -44.84, 2.34) mm, rotated rx 180 ry 0 rz 90 deg; joints [71.546, -19.088, 89.182, 0, 19.905, 71.546]
  MoveL 194 to (-80.02, -45.03, 1.94) mm, rotated rx 180 ry 0 rz 90 deg; joints [71.523, -19.089, 89.265, 0, 19.823, 71.523]
  MoveL 195 to (-81.45, -45.54, 1.53) mm, rotated rx 180 ry 0 rz 90 deg; joints [71.491, -19.087, 89.336, 0, 19.751, 71.491]
  MoveL 196 to (-82.73, -46.35, 1.13) mm, rotated rx -180 ry 0 rz 90 deg; joints [71.449, -19.081, 89.389, 0, 19.692, 71.449]
  MoveL 197 to (-83.8, -47.43, 0.72) mm, rotated rx -180 ry 0 rz 90 deg; joints [71.401, -19.07, 89.423, 0, 19.648, 71.401]
  MoveL 198 to (-84.6, -48.72, 0.31) mm, rotated rx -180 ry 0 rz 90 deg; joints [71.35, -19.055, 89.434, 0, 19.621, 71.35]
  MoveL 199 to (-85.1, -50.16, -0.09) mm, rotated rx -180 ry 0 rz 90 deg; joints [71.296, -19.034, 89.421, 0, 19.613, 71.296]
  MoveL 200 to (-85.24, -51.67, -0.5) mm, rotated rx 180 ry 0 rz 90 deg; joints [71.245, -19.007, 89.383, 0, 19.624, 71.245]
  MoveL 201 to (-85.24, -70.94, -0.5) mm, rotated rx -180 ry 0 rz 90 deg; joints [70.608, -18.905, 88.94, 0, 19.965, 70.608]
  MoveC 202 to (-81.2, -80.65, -0.5) mm, rotated rx -180 ry 0 rz 90 deg; joints [70.337, -18.789, 88.441, 0, 20.348, 70.337] to (-71.47, -84.61, -0.5) mm, rotated rx 180 ry 0 rz 90 deg; joints [70.321, -18.611, 87.694, 0, 20.917, 70.321]
  MoveL 203 to (-35.27, -84.33, -0.5) mm, rotated rx 180 ry 0 rz 90 deg; joints [70.742, -17.999, 85.232, 0, 22.767, 70.742]
  MoveC 204 to (-26.89, -81.41, -0.5) mm, rotated rx -180 ry 0 rz 90 deg; joints [70.928, -17.866, 84.72, 0, 23.146, 70.928] to (-22.01, -74, -0.5) mm, rotated rx -180 ry 0 rz 90 deg; joints [71.217, -17.824, 84.557, 0, 23.266, 71.217]
  MoveL 205 to (-9.28, -25.11, -0.5) mm, rotated rx 180 ry 0 rz 90 deg; joints [72.915, -17.88, 84.774, 0, 23.106, 72.915]
  MoveL 206 to (-8.99, -23.57, -0.5) mm, rotated rx -180 ry 0 rz 90 deg; joints [72.968, -17.884, 84.787, 0, 23.097, 72.968]
  MoveC 207 to (-12.57, -11.97, -0.5) mm, rotated rx 180 ry 0 rz 90 deg; joints [73.308, -18.012, 85.286, 0, 22.727, 73.308] to (-24.15, -8.32, -0.5) mm, rotated rx 180 ry 0 rz 90 deg; joints [73.314, -18.237, 86.171, 0, 22.066, 73.314]
  MoveL 208 to (-25.11, -8.49, -0.5) mm, rotated rx -180 ry 0 rz 90 deg; joints [73.298, -18.253, 86.235, 0, 22.018, 73.298]
  MoveL 209 to (-74.37, -18.97, -0.5) mm, rotated rx 180 ry 0 rz 90 deg; joints [72.451, -19.005, 89.373, 0, 19.632, 72.451]
  MoveC 210 to (-82.18, -23.76, -0.5) mm, rotated rx -180 ry 0 rz 90 deg; joints [72.208, -19.1, 89.792, 0, 19.308, 72.208] to (-85.24, -32.39, -0.5) mm, rotated rx 180 ry 0 rz 90 deg; joints [71.886, -19.104, 89.809, 0, 19.294, 71.886]
  MoveL 211 to (-85.24, -51.67, -0.5) mm, rotated rx 180 ry 0 rz 90 deg; joints [71.245, -19.007, 89.383, 0, 19.624, 71.245]
  MoveL 212 to (-77.69, -51.67, -0.5) mm, rotated rx 180 ry 0 rz 90 deg; joints [71.329, -18.891, 88.88, 0, 20.012, 71.329]
  MoveL 213 to (-77.69, -51.67, 2.5) mm, rotated rx 180 ry 0 rz 90 deg; joints [71.329, -19.047, 88.98, 0, 20.068, 71.329]
  Establecer velocidad (1000.0 mm/s)
  MoveL 214 to (-77.69, -51.67, 10) mm, rotated rx 180 ry 0 rz 90 deg; joints [71.329, -19.438, 89.229, 0, 20.209, 71.329]
  Establecer velocidad (66.7 mm/s)
  MoveL 215 to (19.34, -76.09, 10) mm, rotated rx -180 ry 0 rz 90 deg; joints [71.59, -17.544, 81.915, 0, 25.629, 71.59]
  MoveL 216 to (19.34, -76.09, 2.75) mm, rotated rx -180 ry 0 rz 90 deg; joints [71.59, -17.178, 81.673, 0, 25.505, 71.59]
  MoveL 217 to (19.17, -77.59, 2.34) mm, rotated rx -180 ry 0 rz 90 deg; joints [71.541, -17.151, 81.636, 0, 25.515, 71.541]
  MoveL 218 to (19.37, -79.1, 1.94) mm, rotated rx -180 ry 0 rz 90 deg; joints [71.496, -17.116, 81.571, 0, 25.545, 71.496]
  MoveL 219 to (19.9, -80.53, 1.53) mm, rotated rx -180 ry 0 rz 90 deg; joints [71.458, -17.075, 81.485, 0, 25.591, 71.458]
  MoveL 220 to (20.73, -81.8, 1.13) mm, rotated rx 180 ry 0 rz 90 deg; joints [71.427, -17.029, 81.38, 0, 25.649, 71.427]
  MoveL 221 to (21.82, -82.85, 0.72) mm, rotated rx 180 ry 0 rz 90 deg; joints [71.405, -16.979, 81.261, 0, 25.718, 71.405]
  MoveL 222 to (23.12, -83.65, 0.31) mm, rotated rx 180 ry 0 rz 90 deg; joints [71.394, -16.927, 81.134, 0, 25.793, 71.394]
  MoveL 223 to (24.56, -84.13, -0.09) mm, rotated rx -180 ry 0 rz 90 deg; joints [71.394, -16.873, 81.004, 0, 25.87, 71.394]
  MoveL 224 to (26.07, -84.25, -0.5) mm, rotated rx -180 ry 0 rz 90 deg; joints [71.406, -16.821, 80.877, 0, 25.944, 71.406]
  MoveL 225 to (53.54, -83.96, -0.5) mm, rotated rx -180 ry 0 rz 90 deg; joints [71.697, -16.237, 78.856, 0, 27.382, 71.697]
  MoveL 226 to (55.92, -83.78, -0.5) mm, rotated rx -180 ry 0 rz 90 deg; joints [71.727, -16.186, 78.682, 0, 27.504, 71.727]
  MoveC 227 to (62, -81.49, -0.5) mm, rotated rx 180 ry 0 rz 90 deg; joints [71.858, -16.068, 78.282, 0, 27.786, 71.858] to (65.88, -76.29, -0.5) mm, rotated rx 180 ry 0 rz 90 deg; joints [72.055, -16.019, 78.117, 0, 27.902, 72.055]
  MoveC 228 to (66.02, -70.36, -0.5) mm, rotated rx 180 ry 0 rz 90 deg; joints [72.237, -16.059, 78.251, 0, 27.808, 72.237] to (63.49, -65, -0.5) mm, rotated rx 180 ry 0 rz 90 deg; joints [72.377, -16.153, 78.57, 0, 27.583, 72.377]
  MoveL 229 to (61.92, -63.02, -0.5) mm, rotated rx -180 ry 0 rz 90 deg; joints [72.422, -16.202, 78.736, 0, 27.466, 72.422]
  MoveL 230 to (33.64, -30.34, -0.5) mm, rotated rx 180 ry 0 rz 90 deg; joints [73.166, -17.019, 81.581, 0, 25.438, 73.166]
  MoveL 231 to (32.69, -29.3, -0.5) mm, rotated rx 180 ry 0 rz 90 deg; joints [73.189, -17.045, 81.673, 0, 25.371, 73.189]
  MoveL 232 to (31.75, -28.42, -0.5) mm, rotated rx 180 ry 0 rz 90 deg; joints [73.208, -17.069, 81.762, 0, 25.308, 73.208]
  MoveL 233 to (16.58, -16.32, -0.5) mm, rotated rx 180 ry 0 rz 90 deg; joints [73.447, -17.442, 83.122, 0, 24.32, 73.447]
  MoveL 234 to (15.64, -15.68, -0.5) mm, rotated rx 180 ry 0 rz 90 deg; joints [73.459, -17.464, 83.204, 0, 24.26, 73.459]
  MoveC 235 to (4.61, -14.15, -0.5) mm, rotated rx -180 ry 0 rz 90 deg; joints [73.403, -17.684, 84.026, 0, 23.658, 73.403] to (-3.01, -22.27, -0.5) mm, rotated rx -180 ry 0 rz 90 deg; joints [73.068, -17.781, 84.393, 0, 23.388, 73.068]
  MoveL 236 to (-15.44, -68.95, -0.5) mm, rotated rx 180 ry 0 rz 90 deg; joints [71.449, -17.734, 84.216, 0, 23.518, 71.449]
  MoveC 237 to (-13.39, -79.56, -0.5) mm, rotated rx -180 ry 0 rz 90 deg; joints [71.134, -17.629, 83.819, 0, 23.81, 71.134] to (-3.79, -84.52, -0.5) mm, rotated rx 180 ry 0 rz 90 deg; joints [71.081, -17.414, 83.019, 0, 24.395, 71.081]
  MoveL 238 to (-2.37, -84.56, -0.5) mm, rotated rx 180 ry 0 rz 90 deg; joints [71.095, -17.387, 82.917, 0, 24.469, 71.095]
  MoveL 239 to (26.07, -84.25, -0.5) mm, rotated rx -180 ry 0 rz 90 deg; joints [71.406, -16.821, 80.877, 0, 25.944, 71.406]
  MoveL 240 to (25.99, -76.7, -0.5) mm, rotated rx 180 ry 0 rz 90 deg; joints [71.64, -16.874, 81.066, 0, 25.808, 71.64]
  MoveL 241 to (25.99, -76.7, 2.5) mm, rotated rx 180 ry 0 rz 90 deg; joints [71.64, -17.026, 81.167, 0, 25.858, 71.64]
  Establecer velocidad (1000.0 mm/s)
  MoveL 242 to (25.99, -76.7, 10) mm, rotated rx 180 ry 0 rz 90 deg; joints [71.64, -17.404, 81.417, 0, 25.986, 71.64]
  Establecer velocidad (66.7 mm/s)
  MoveL 243 to (74.55, -31.86, 10) mm, rotated rx 180 ry 0 rz 90 deg; joints [73.5, -16.658, 78.857, 0, 27.802, 73.5]
  MoveL 244 to (74.55, -31.86, 2.75) mm, rotated rx 180 ry 0 rz 90 deg; joints [73.5, -16.296, 78.614, 0, 27.682, 73.5]
  MoveL 245 to (76.06, -32.04, 2.34) mm, rotated rx -180 ry 0 rz 90 deg; joints [73.508, -16.241, 78.482, 0, 27.759, 73.508]
  MoveL 246 to (77.56, -31.86, 1.94) mm, rotated rx 180 ry 0 rz 90 deg; joints [73.527, -16.188, 78.357, 0, 27.83, 73.527]
  MoveL 247 to (78.99, -31.34, 1.53) mm, rotated rx 180 ry 0 rz 90 deg; joints [73.556, -16.138, 78.247, 0, 27.892, 73.556]
  MoveL 248 to (80.28, -30.53, 1.13) mm, rotated rx 180 ry 0 rz 90 deg; joints [73.593, -16.094, 78.153, 0, 27.941, 73.593]
  MoveL 249 to (81.35, -29.45, 0.72) mm, rotated rx -180 ry 0 rz 90 deg; joints [73.636, -16.057, 78.082, 0, 27.975, 73.636]
  MoveL 250 to (82.15, -28.16, 0.31) mm, rotated rx 180 ry 0 rz 90 deg; joints [73.682, -16.027, 78.036, 0, 27.991, 73.682]
  MoveL 251 to (82.65, -26.72, -0.09) mm, rotated rx 180 ry 0 rz 90 deg; joints [73.731, -16.005, 78.016, 0, 27.989, 73.731]
  MoveL 252 to (82.79, -25.21, -0.5) mm, rotated rx -180 ry 0 rz 90 deg; joints [73.779, -15.991, 78.026, 0, 27.966, 73.779]
  MoveL 253 to (82.78, -4.26, -0.5) mm, rotated rx 180 ry 0 rz 90 deg; joints [74.425, -16.127, 78.481, 0, 27.646, 74.425]
  MoveL 254 to (82.69, -1.88, -0.5) mm, rotated rx -180 ry 0 rz 90 deg; joints [74.498, -16.144, 78.538, 0, 27.605, 74.498]
  MoveC 255 to (81.43, 3.51, -0.5) mm, rotated rx 180 ry 0 rz 90 deg; joints [74.655, -16.205, 78.747, 0, 27.458, 74.655] to (78.27, 8.05, -0.5) mm, rotated rx -180 ry 0 rz 90 deg; joints [74.769, -16.304, 79.081, 0, 27.222, 74.769]
  MoveC 256 to (71.54, 10.15, -0.5) mm, rotated rx 180 ry 0 rz 90 deg; joints [74.777, -16.464, 79.633, 0, 26.831, 74.777] to (65.09, 7.29, -0.5) mm, rotated rx 180 ry 0 rz 90 deg; joints [74.633, -16.587, 80.058, 0, 26.529, 74.633]
  MoveC 257 to (62.39, 4.4, -0.5) mm, rotated rx -180 ry 0 rz 90 deg; joints [74.519, -16.628, 80.201, 0, 26.427, 74.519] to (59.93, 1.3, -0.5) mm, rotated rx 180 ry 0 rz 90 deg; joints [74.4, -16.662, 80.32, 0, 26.342, 74.4]
  MoveL 258 to (45.5, -18.48, -0.5) mm, rotated rx 180 ry 0 rz 90 deg; joints [73.65, -16.847, 80.97, 0, 25.877, 73.65]
  MoveL 259 to (44.97, -19.24, -0.5) mm, rotated rx -180 ry 0 rz 90 deg; joints [73.621, -16.854, 80.992, 0, 25.861, 73.621]
  MoveC 260 to (42.84, -26.7, -0.5) mm, rotated rx -180 ry 0 rz 90 deg; joints [73.367, -16.852, 80.986, 0, 25.865, 73.367] to (45.8, -33.88, -0.5) mm, rotated rx -180 ry 0 rz 90 deg; joints [73.17, -16.745, 80.609, 0, 26.135, 73.17]
  MoveL 261 to (62.07, -52.28, -0.5) mm, rotated rx 180 ry 0 rz 90 deg; joints [72.754, -16.273, 78.978, 0, 27.296, 72.754]
  MoveL 262 to (63.62, -53.88, -0.5) mm, rotated rx 180 ry 0 rz 90 deg; joints [72.719, -16.228, 78.824, 0, 27.404, 72.719]
  MoveC 263 to (68.57, -57, -0.5) mm, rotated rx 180 ry 0 rz 90 deg; joints [72.671, -16.096, 78.378, 0, 27.718, 72.671] to (74.39, -57.5, -0.5) mm, rotated rx 180 ry 0 rz 90 deg; joints [72.711, -15.961, 77.925, 0, 28.037, 72.711]
  MoveC 264 to (79.66, -54.17, -0.5) mm, rotated rx -180 ry 0 rz 90 deg; joints [72.863, -15.865, 77.602, 0, 28.263, 72.863] to (82.25, -48.51, -0.5) mm, rotated rx -180 ry 0 rz 90 deg; joints [73.06, -15.845, 77.537, 0, 28.308, 73.06]
  MoveL 265 to (82.74, -45.01, -0.5) mm, rotated rx -180 ry 0 rz 90 deg; joints [73.171, -15.858, 77.58, 0, 28.278, 73.171]
  MoveL 266 to (82.78, -44.07, -0.5) mm, rotated rx 180 ry 0 rz 90 deg; joints [73.2, -15.864, 77.599, 0, 28.264, 73.2]
  MoveL 267 to (82.79, -43.12, -0.5) mm, rotated rx -180 ry 0 rz 90 deg; joints [73.23, -15.87, 77.62, 0, 28.25, 73.23]
  MoveL 268 to (82.79, -25.21, -0.5) mm, rotated rx -180 ry 0 rz 90 deg; joints [73.779, -15.991, 78.026, 0, 27.966, 73.779]
  MoveL 269 to (75.24, -25.21, -0.5) mm, rotated rx -180 ry 0 rz 90 deg; joints [73.711, -16.162, 78.6, 0, 27.562, 73.711]
  MoveL 270 to (75.24, -25.21, 2.5) mm, rotated rx 180 ry 0 rz 90 deg; joints [73.711, -16.312, 78.701, 0, 27.611, 73.711]
  Establecer velocidad (1000.0 mm/s)
  MoveL 271 to (75.24, -25.21, 10) mm, rotated rx 180 ry 0 rz 90 deg; joints [73.711, -16.687, 78.953, 0, 27.734, 73.711]
  Establecer velocidad (66.7 mm/s)
  MoveL 272 to (37.86, 31.84, 10) mm, rotated rx -180 ry 0 rz 90 deg; joints [75.178, -17.822, 82.911, 0, 24.911, 75.178]
  MoveL 273 to (37.86, 31.84, 2.75) mm, rotated rx -180 ry 0 rz 90 deg; joints [75.178, -17.455, 82.67, 0, 24.785, 75.178]
  MoveL 274 to (38, 33.35, 2.34) mm, rotated rx 180 ry 0 rz 90 deg; joints [75.227, -17.439, 82.675, 0, 24.764, 75.227]
  MoveL 275 to (37.77, 34.86, 1.94) mm, rotated rx -180 ry 0 rz 90 deg; joints [75.273, -17.431, 82.707, 0, 24.724, 75.273]
  MoveL 276 to (37.22, 36.27, 1.53) mm, rotated rx 180 ry 0 rz 90 deg; joints [75.314, -17.429, 82.76, 0, 24.668, 75.314]
  MoveL 277 to (36.37, 37.53, 1.13) mm, rotated rx 180 ry 0 rz 90 deg; joints [75.347, -17.431, 82.833, 0, 24.599, 75.347]
  MoveL 278 to (35.27, 38.57, 0.72) mm, rotated rx 180 ry 0 rz 90 deg; joints [75.372, -17.438, 82.92, 0, 24.519, 75.372]
  MoveL 279 to (33.95, 39.34, 0.31) mm, rotated rx 180 ry 0 rz 90 deg; joints [75.385, -17.447, 83.016, 0, 24.431, 75.385]
  MoveL 280 to (32.51, 39.8, -0.09) mm, rotated rx 180 ry 0 rz 90 deg; joints [75.388, -17.458, 83.116, 0, 24.341, 75.388]
  MoveL 281 to (30.99, 39.9, -0.5) mm, rotated rx 180 ry 0 rz 90 deg; joints [75.378, -17.467, 83.214, 0, 24.253, 75.378]
  MoveL 282 to (7.11, 39.25, -0.5) mm, rotated rx -180 ry 0 rz 90 deg; joints [75.154, -17.917, 84.917, 0, 23, 75.154]
  MoveL 283 to (6.16, 39.16, -0.5) mm, rotated rx 180 ry 0 rz 90 deg; joints [75.143, -17.934, 84.983, 0, 22.951, 75.143]
  MoveC 284 to (-2.98, 33.75, -0.5) mm, rotated rx 180 ry 0 rz 90 deg; joints [74.886, -18.074, 85.528, 0, 22.547, 74.886] to (-4.29, 23.22, -0.5) mm, rotated rx 180 ry 0 rz 90 deg; joints [74.53, -18.046, 85.417, 0, 22.629, 74.53]
  MoveL 285 to (-3.98, 22.27, -0.5) mm, rotated rx 180 ry 0 rz 90 deg; joints [74.502, -18.036, 85.377, 0, 22.659, 74.502]
  MoveL 286 to (1.87, 6.16, -0.5) mm, rotated rx -180 ry 0 rz 90 deg; joints [74.032, -17.846, 84.642, 0, 23.204, 74.032]
  MoveL 287 to (2.33, 5.02, -0.5) mm, rotated rx -180 ry 0 rz 90 deg; joints [73.999, -17.831, 84.586, 0, 23.245, 73.999]
  MoveC 288 to (3.9, 2.25, -0.5) mm, rotated rx -180 ry 0 rz 90 deg; joints [73.924, -17.787, 84.418, 0, 23.369, 73.924] to (6.13, -0.02, -0.5) mm, rotated rx 180 ry 0 rz 90 deg; joints [73.872, -17.733, 84.213, 0, 23.521, 73.872]
  MoveL 289 to (23.22, -13.31, -0.5) mm, rotated rx 180 ry 0 rz 90 deg; joints [73.606, -17.33, 82.708, 0, 24.622, 73.606]
  MoveL 290 to (23.8, -13.74, -0.5) mm, rotated rx 180 ry 0 rz 90 deg; joints [73.598, -17.316, 82.657, 0, 24.659, 73.598]
  MoveC 291 to (33.06, -15.98, -0.5) mm, rotated rx 180 ry 0 rz 90 deg; joints [73.613, -17.118, 81.936, 0, 25.182, 73.613] to (41.13, -10.9, -0.5) mm, rotated rx 180 ry 0 rz 90 deg; joints [73.848, -16.983, 81.455, 0, 25.529, 73.848]
  MoveL 292 to (63.57, 20.37, -0.5) mm, rotated rx 180 ry 0 rz 90 deg; joints [75.031, -16.696, 80.437, 0, 26.259, 75.031]
  MoveL 293 to (64.63, 21.89, -0.5) mm, rotated rx 180 ry 0 rz 90 deg; joints [75.087, -16.682, 80.388, 0, 26.293, 75.087]
  MoveC 294 to (66.87, 27.57, -0.5) mm, rotated rx 180 ry 0 rz 90 deg; joints [75.285, -16.666, 80.333, 0, 26.333, 75.285] to (66.35, 33.64, -0.5) mm, rotated rx -180 ry 0 rz 90 deg; joints [75.472, -16.711, 80.49, 0, 26.221, 75.472]
  MoveC 295 to (62.06, 38.56, -0.5) mm, rotated rx 180 ry 0 rz 90 deg; joints [75.592, -16.829, 80.905, 0, 25.924, 75.592] to (55.83, 40.47, -0.5) mm, rotated rx -180 ry 0 rz 90 deg; joints [75.602, -16.97, 81.405, 0, 25.565, 75.602]
  MoveL 296 to (53.54, 40.52, -0.5) mm, rotated rx 180 ry 0 rz 90 deg; joints [75.585, -17.017, 81.575, 0, 25.442, 75.585]
  MoveL 297 to (30.99, 39.9, -0.5) mm, rotated rx 180 ry 0 rz 90 deg; joints [75.378, -17.467, 83.214, 0, 24.253, 75.378]
  MoveL 298 to (31.2, 32.35, -0.5) mm, rotated rx -180 ry 0 rz 90 deg; joints [75.137, -17.424, 83.055, 0, 24.369, 75.137]
  MoveL 299 to (31.2, 32.35, 2.5) mm, rotated rx -180 ry 0 rz 90 deg; joints [75.137, -17.577, 83.156, 0, 24.421, 75.137]
  Establecer velocidad (1000.0 mm/s)
  MoveL 300 to (31.2, 32.35, 10) mm, rotated rx -180 ry 0 rz 90 deg; joints [75.137, -17.957, 83.405, 0, 24.552, 75.137]
  Establecer velocidad (66.7 mm/s)
  MoveL 301 to (26.12, 75.73, 10) mm, rotated rx -180 ry 0 rz 90 deg; joints [76.5, -18.269, 84.565, 0, 23.705, 76.5]
  MoveL 302 to (26.12, 75.73, 2.75) mm, rotated rx 180 ry 0 rz 90 deg; joints [76.5, -17.9, 84.324, 0, 23.576, 76.5]
  MoveL 303 to (26.33, 77.24, 2.34) mm, rotated rx -180 ry 0 rz 90 deg; joints [76.551, -17.882, 84.322, 0, 23.56, 76.551]
  MoveL 304 to (26.16, 78.75, 1.94) mm, rotated rx 180 ry 0 rz 90 deg; joints [76.599, -17.871, 84.346, 0, 23.525, 76.599]
  MoveL 305 to (25.67, 80.18, 1.53) mm, rotated rx -180 ry 0 rz 90 deg; joints [76.642, -17.866, 84.393, 0, 23.474, 76.642]
  MoveL 306 to (24.87, 81.48, 1.13) mm, rotated rx -180 ry 0 rz 90 deg; joints [76.678, -17.867, 84.459, 0, 23.408, 76.678]
  MoveL 307 to (23.8, 82.56, 0.72) mm, rotated rx 180 ry 0 rz 90 deg; joints [76.705, -17.871, 84.54, 0, 23.33, 76.705]
  MoveL 308 to (22.52, 83.38, 0.31) mm, rotated rx 180 ry 0 rz 90 deg; joints [76.722, -17.878, 84.633, 0, 23.245, 76.722]
  MoveL 309 to (21.09, 83.9, -0.09) mm, rotated rx -180 ry 0 rz 90 deg; joints [76.728, -17.886, 84.73, 0, 23.156, 76.728]
  MoveL 310 to (19.59, 84.05, -0.5) mm, rotated rx -180 ry 0 rz 90 deg; joints [76.722, -17.894, 84.828, 0, 23.066, 76.722]
  MoveL 311 to (-29.85, 84.67, -0.5) mm, rotated rx -180 ry 0 rz 90 deg; joints [76.348, -18.759, 88.313, 0, 20.446, 76.348]
  MoveL 312 to (-32.6, 84.59, -0.5) mm, rotated rx -180 ry 0 rz 90 deg; joints [76.323, -18.803, 88.501, 0, 20.302, 76.323]
  MoveC 313 to (-37.67, 83.81, -0.5) mm, rotated rx -180 ry 0 rz 90 deg; joints [76.255, -18.881, 88.836, 0, 20.045, 76.255] to (-42.39, 81.78, -0.5) mm, rotated rx -180 ry 0 rz 90 deg; joints [76.147, -18.948, 89.125, 0, 19.823, 76.147]
  MoveC 314 to (-47.09, 74.96, -0.5) mm, rotated rx 180 ry 0 rz 90 deg; joints [75.876, -18.995, 89.33, 0, 19.665, 75.876] to (-44.92, 66.96, -0.5) mm, rotated rx -180 ry 0 rz 90 deg; joints [75.624, -18.929, 89.043, 0, 19.886, 75.624]
  MoveC 315 to (-41.77, 63.75, -0.5) mm, rotated rx -180 ry 0 rz 90 deg; joints [75.543, -18.866, 88.771, 0, 20.095, 75.543] to (-38.16, 61.06, -0.5) mm, rotated rx 180 ry 0 rz 90 deg; joints [75.483, -18.797, 88.477, 0, 20.32, 75.483]
  MoveL 316 to (-15.91, 46.95, -0.5) mm, rotated rx 180 ry 0 rz 90 deg; joints [75.207, -18.364, 86.682, 0, 21.682, 75.207]
  MoveC 317 to (-11.3, 44.97, -0.5) mm, rotated rx 180 ry 0 rz 90 deg; joints [75.182, -18.275, 86.323, 0, 21.952, 75.182] to (-6.3, 44.55, -0.5) mm, rotated rx 180 ry 0 rz 90 deg; joints [75.211, -18.185, 85.965, 0, 22.22, 75.211]
  MoveL 318 to (-0.15, 45.01, -0.5) mm, rotated rx 180 ry 0 rz 90 deg; joints [75.28, -18.077, 85.54, 0, 22.537, 75.28]
  MoveL 319 to (65.45, 49.75, -0.5) mm, rotated rx -180 ry 0 rz 90 deg; joints [75.975, -16.817, 80.864, 0, 25.953, 75.975]
  MoveL 320 to (72.21, 50.17, -0.5) mm, rotated rx -180 ry 0 rz 90 deg; joints [76.041, -16.675, 80.365, 0, 26.31, 76.041]
  MoveC 321 to (79.24, 53.37, -0.5) mm, rotated rx 180 ry 0 rz 90 deg; joints [76.197, -16.54, 79.895, 0, 26.645, 76.197] to (82.34, 60.45, -0.5) mm, rotated rx 180 ry 0 rz 90 deg; joints [76.444, -16.51, 79.792, 0, 26.719, 76.444]
  MoveL 322 to (82.37, 61.12, -0.5) mm, rotated rx -180 ry 0 rz 90 deg; joints [76.465, -16.513, 79.802, 0, 26.712, 76.465]
  MoveL 323 to (82.36, 72.49, -0.5) mm, rotated rx 180 ry 0 rz 90 deg; joints [76.825, -16.572, 80.006, 0, 26.566, 76.825]
  MoveL 324 to (82.33, 73.05, -0.5) mm, rotated rx 180 ry 0 rz 90 deg; joints [76.842, -16.576, 80.019, 0, 26.557, 76.842]
  MoveC 325 to (79.04, 80.2, -0.5) mm, rotated rx 180 ry 0 rz 90 deg; joints [77.044, -16.683, 80.393, 0, 26.29, 77.044] to (71.77, 83.23, -0.5) mm, rotated rx 180 ry 0 rz 90 deg; joints [77.088, -16.853, 80.991, 0, 25.862, 77.088]
  MoveL 326 to (54.49, 83.62, -0.5) mm, rotated rx -180 ry 0 rz 90 deg; joints [76.973, -17.213, 82.282, 0, 24.931, 76.973]
  MoveL 327 to (19.59, 84.05, -0.5) mm, rotated rx -180 ry 0 rz 90 deg; joints [76.722, -17.894, 84.828, 0, 23.066, 76.722]
  MoveL 328 to (19.49, 76.5, -0.5) mm, rotated rx 180 ry 0 rz 90 deg; joints [76.474, -17.862, 84.705, 0, 23.157, 76.474]
  MoveL 329 to (19.49, 76.5, 2.5) mm, rotated rx 180 ry 0 rz 90 deg; joints [76.474, -18.016, 84.806, 0, 23.21, 76.474]
  Establecer velocidad (1000.0 mm/s)
  MoveL 330 to (19.49, 76.5, 10) mm, rotated rx 180 ry 0 rz 90 deg; joints [76.474, -18.399, 85.055, 0, 23.344, 76.474]
  Establecer velocidad (66.7 mm/s)
  MoveL 331 to (26.1, 74.91, 10) mm, rotated rx -180 ry 0 rz 90 deg; joints [76.473, -18.266, 84.552, 0, 23.714, 76.473]
  MoveL 332 to (26.1, 74.91, 2.5) mm, rotated rx 180 ry 0 rz 90 deg; joints [76.473, -17.884, 84.303, 0, 23.58, 76.473]
  MoveL 333 to (26.31, 76.41, 2.09) mm, rotated rx -180 ry 0 rz 90 deg; joints [76.524, -17.866, 84.301, 0, 23.565, 76.524]
  MoveL 334 to (26.14, 77.92, 1.69) mm, rotated rx -180 ry 0 rz 90 deg; joints [76.572, -17.855, 84.325, 0, 23.53, 76.572]
  MoveL 335 to (25.65, 79.36, 1.28) mm, rotated rx 180 ry 0 rz 90 deg; joints [76.615, -17.85, 84.372, 0, 23.479, 76.615]
  MoveL 336 to (24.85, 80.66, 0.87) mm, rotated rx -180 ry 0 rz 90 deg; joints [76.651, -17.85, 84.438, 0, 23.413, 76.651]
  MoveL 337 to (23.79, 81.74, 0.47) mm, rotated rx 180 ry 0 rz 90 deg; joints [76.678, -17.855, 84.519, 0, 23.336, 76.678]
  MoveL 338 to (22.51, 82.56, 0.06) mm, rotated rx -180 ry 0 rz 90 deg; joints [76.695, -17.862, 84.611, 0, 23.25, 76.695]
  MoveL 339 to (21.08, 83.08, -0.34) mm, rotated rx 180 ry 0 rz 90 deg; joints [76.701, -17.87, 84.709, 0, 23.161, 76.701]
  MoveL 340 to (19.58, 83.24, -0.75) mm, rotated rx 180 ry 0 rz 90 deg; joints [76.695, -17.878, 84.806, 0, 23.072, 76.695]
  MoveC 341 to (-5.61, 83.54, -0.75) mm, rotated rx -180 ry 0 rz 90 deg; joints [76.507, -18.333, 86.599, 0, 21.734, 76.507] to (-30.8, 83.73, -0.75) mm, rotated rx 180 ry 0 rz 90 deg; joints [76.309, -18.757, 88.354, 0, 20.403, 76.309]
  MoveC 342 to (-36.14, 83.21, -0.75) mm, rotated rx -180 ry 0 rz 90 deg; joints [76.247, -18.841, 88.713, 0, 20.129, 76.247] to (-41.22, 81.46, -0.75) mm, rotated rx -180 ry 0 rz 90 deg; joints [76.146, -18.915, 89.031, 0, 19.884, 76.146]
  MoveC 343 to (-45.93, 75.9, -0.75) mm, rotated rx 180 ry 0 rz 90 deg; joints [75.918, -18.967, 89.258, 0, 19.709, 75.918] to (-44.91, 68.69, -0.75) mm, rotated rx 180 ry 0 rz 90 deg; joints [75.682, -18.923, 89.064, 0, 19.859, 75.682]
  MoveC 344 to (-42.16, 65.24, -0.75) mm, rotated rx -180 ry 0 rz 90 deg; joints [75.589, -18.866, 88.817, 0, 20.049, 75.589] to (-38.73, 62.49, -0.75) mm, rotated rx 180 ry 0 rz 90 deg; joints [75.526, -18.799, 88.533, 0, 20.267, 75.526]
  MoveL 345 to (-15.64, 47.86, -0.75) mm, rotated rx -180 ry 0 rz 90 deg; joints [75.239, -18.351, 86.672, 0, 21.679, 75.239]
  MoveL 346 to (-14.99, 47.48, -0.75) mm, rotated rx 180 ry 0 rz 90 deg; joints [75.232, -18.338, 86.62, 0, 21.718, 75.232]
  MoveC 347 to (-10.87, 45.81, -0.75) mm, rotated rx 180 ry 0 rz 90 deg; joints [75.213, -18.259, 86.301, 0, 21.958, 75.213] to (-6.44, 45.46, -0.75) mm, rotated rx 180 ry 0 rz 90 deg; joints [75.24, -18.179, 85.983, 0, 22.196, 75.24]
  MoveL 348 to (72.49, 51.11, -0.75) mm, rotated rx -180 ry 0 rz 90 deg; joints [76.073, -16.662, 80.354, 0, 26.308, 76.073]
  MoveC 349 to (78.6, 54.02, -0.75) mm, rotated rx 180 ry 0 rz 90 deg; joints [76.212, -16.545, 79.948, 0, 26.597, 76.212] to (81.39, 60.18, -0.75) mm, rotated rx -180 ry 0 rz 90 deg; joints [76.428, -16.517, 79.85, 0, 26.667, 76.428]
  MoveL 350 to (81.44, 61.12, -0.75) mm, rotated rx -180 ry 0 rz 90 deg; joints [76.458, -16.521, 79.864, 0, 26.657, 76.458]
  MoveL 351 to (81.43, 72.49, -0.75) mm, rotated rx -180 ry 0 rz 90 deg; joints [76.818, -16.58, 80.068, 0, 26.512, 76.818]
  MoveL 352 to (81.39, 73.13, -0.75) mm, rotated rx -180 ry 0 rz 90 deg; joints [76.837, -16.584, 80.083, 0, 26.501, 76.837]
  MoveC 353 to (78.36, 79.57, -0.75) mm, rotated rx -180 ry 0 rz 90 deg; joints [77.02, -16.682, 80.424, 0, 26.258, 77.02] to (71.78, 82.3, -0.75) mm, rotated rx -180 ry 0 rz 90 deg; joints [77.058, -16.836, 80.966, 0, 25.87, 77.058]
  MoveC 354 to (45.68, 82.82, -0.75) mm, rotated rx 180 ry 0 rz 90 deg; joints [76.881, -17.374, 82.908, 0, 24.466, 76.881] to (19.58, 83.24, -0.75) mm, rotated rx 180 ry 0 rz 90 deg; joints [76.695, -17.878, 84.806, 0, 23.072, 76.695]
  MoveL 355 to (19.47, 75.69, -0.75) mm, rotated rx 180 ry 0 rz 90 deg; joints [76.447, -17.846, 84.685, 0, 23.162, 76.447]
  MoveL 356 to (19.47, 75.69, 2.25) mm, rotated rx 180 ry 0 rz 90 deg; joints [76.447, -18, 84.785, 0, 23.215, 76.447]
  Establecer velocidad (1000.0 mm/s)
  MoveL 357 to (19.47, 75.69, 10) mm, rotated rx -180 ry 0 rz 90 deg; joints [76.447, -18.396, 85.042, 0, 23.353, 76.447]
  Establecer velocidad (66.7 mm/s)
  MoveL 358 to (37.75, 30.9, 10) mm, rotated rx -180 ry 0 rz 90 deg; joints [75.146, -17.819, 82.9, 0, 24.919, 75.146]
  MoveL 359 to (37.75, 30.9, 2.5) mm, rotated rx 180 ry 0 rz 90 deg; joints [75.146, -17.439, 82.651, 0, 24.788, 75.146]
  MoveL 360 to (37.9, 32.41, 2.09) mm, rotated rx -180 ry 0 rz 90 deg; joints [75.196, -17.423, 82.656, 0, 24.768, 75.196]
  MoveL 361 to (37.67, 33.91, 1.69) mm, rotated rx 180 ry 0 rz 90 deg; joints [75.242, -17.415, 82.688, 0, 24.728, 75.242]
  MoveL 362 to (37.12, 35.33, 1.28) mm, rotated rx 180 ry 0 rz 90 deg; joints [75.283, -17.413, 82.741, 0, 24.672, 75.283]
  MoveL 363 to (36.27, 36.59, 0.87) mm, rotated rx -180 ry 0 rz 90 deg; joints [75.316, -17.416, 82.814, 0, 24.602, 75.316]
  MoveL 364 to (35.16, 37.63, 0.47) mm, rotated rx 180 ry 0 rz 90 deg; joints [75.34, -17.423, 82.901, 0, 24.522, 75.34]
  MoveL 365 to (33.85, 38.4, 0.06) mm, rotated rx 180 ry 0 rz 90 deg; joints [75.354, -17.432, 82.997, 0, 24.435, 75.354]
  MoveL 366 to (32.4, 38.85, -0.34) mm, rotated rx -180 ry 0 rz 90 deg; joints [75.357, -17.442, 83.097, 0, 24.345, 75.357]
  MoveL 367 to (30.89, 38.95, -0.75) mm, rotated rx -180 ry 0 rz 90 deg; joints [75.347, -17.452, 83.195, 0, 24.256, 75.347]
  MoveL 368 to (7.11, 38.3, -0.75) mm, rotated rx 180 ry 0 rz 90 deg; joints [75.123, -17.9, 84.891, 0, 23.009, 75.123]
  MoveL 369 to (5.91, 38.18, -0.75) mm, rotated rx -180 ry 0 rz 90 deg; joints [75.108, -17.921, 84.974, 0, 22.947, 75.108]
  MoveC 370 to (-2.15, 33.35, -0.75) mm, rotated rx 180 ry 0 rz 90 deg; joints [74.88, -18.045, 85.453, 0, 22.591, 74.88] to (-3.55, 24.06, -0.75) mm, rotated rx -180 ry 0 rz 90 deg; joints [74.564, -18.024, 85.373, 0, 22.651, 74.564]
  MoveL 371 to (-3.01, 22.27, -0.75) mm, rotated rx 180 ry 0 rz 90 deg; joints [74.511, -18.005, 85.3, 0, 22.706, 74.511]
  MoveL 372 to (2.9, 6.02, -0.75) mm, rotated rx -180 ry 0 rz 90 deg; joints [74.037, -17.813, 84.557, 0, 23.256, 74.037]
  MoveC 373 to (4.45, 3.1, -0.75) mm, rotated rx 180 ry 0 rz 90 deg; joints [73.957, -17.769, 84.387, 0, 23.381, 73.957] to (6.75, 0.72, -0.75) mm, rotated rx 180 ry 0 rz 90 deg; joints [73.901, -17.713, 84.175, 0, 23.538, 73.901]
  MoveL 374 to (9.47, -1.42, -0.75) mm, rotated rx -180 ry 0 rz 90 deg; joints [73.858, -17.65, 83.937, 0, 23.713, 73.858]
  MoveL 375 to (21.66, -10.9, -0.75) mm, rotated rx 180 ry 0 rz 90 deg; joints [73.668, -17.362, 82.864, 0, 24.498, 73.668]
  MoveL 376 to (24.17, -12.82, -0.75) mm, rotated rx -180 ry 0 rz 90 deg; joints [73.63, -17.301, 82.641, 0, 24.66, 73.63]
  MoveC 377 to (32.44, -15.15, -0.75) mm, rotated rx -180 ry 0 rz 90 deg; joints [73.633, -17.122, 81.991, 0, 25.132, 73.633] to (39.91, -10.9, -0.75) mm, rotated rx 180 ry 0 rz 90 deg; joints [73.837, -16.996, 81.535, 0, 25.461, 73.837]
  MoveL 378 to (40.67, -9.95, -0.75) mm, rotated rx 180 ry 0 rz 90 deg; joints [73.874, -16.986, 81.5, 0, 25.486, 73.874]
  MoveL 379 to (63.73, 22.27, -0.75) mm, rotated rx -180 ry 0 rz 90 deg; joints [75.092, -16.691, 80.455, 0, 26.236, 75.092]
  MoveC 380 to (65.98, 27.75, -0.75) mm, rotated rx 180 ry 0 rz 90 deg; joints [75.283, -16.674, 80.395, 0, 26.279, 75.283] to (65.35, 33.64, -0.75) mm, rotated rx 180 ry 0 rz 90 deg; joints [75.464, -16.72, 80.557, 0, 26.163, 75.464]
  MoveC 381 to (61.41, 37.88, -0.75) mm, rotated rx -180 ry 0 rz 90 deg; joints [75.566, -16.826, 80.932, 0, 25.894, 75.566] to (55.88, 39.56, -0.75) mm, rotated rx 180 ry 0 rz 90 deg; joints [75.574, -16.951, 81.375, 0, 25.576, 75.574]
  MoveL 382 to (54.49, 39.6, -0.75) mm, rotated rx 180 ry 0 rz 90 deg; joints [75.564, -16.98, 81.479, 0, 25.501, 75.564]
  MoveL 383 to (30.89, 38.95, -0.75) mm, rotated rx -180 ry 0 rz 90 deg; joints [75.347, -17.452, 83.195, 0, 24.256, 75.347]
  MoveL 384 to (31.1, 31.4, -0.75) mm, rotated rx -180 ry 0 rz 90 deg; joints [75.106, -17.408, 83.036, 0, 24.373, 75.106]
  MoveL 385 to (31.1, 31.4, 2.25) mm, rotated rx -180 ry 0 rz 90 deg; joints [75.106, -17.561, 83.136, 0, 24.424, 75.106]
  Establecer velocidad (1000.0 mm/s)
  MoveL 386 to (31.1, 31.4, 10) mm, rotated rx 180 ry 0 rz 90 deg; joints [75.106, -17.954, 83.394, 0, 24.56, 75.106]
  Establecer velocidad (66.7 mm/s)
  MoveL 387 to (73.63, -30.54, 10) mm, rotated rx -180 ry 0 rz 90 deg; joints [73.532, -16.688, 78.956, 0, 27.732, 73.532]
  MoveL 388 to (73.63, -30.54, 2.5) mm, rotated rx -180 ry 0 rz 90 deg; joints [73.532, -16.313, 78.704, 0, 27.609, 73.532]
  MoveL 389 to (75.14, -30.73, 2.09) mm, rotated rx 180 ry 0 rz 90 deg; joints [73.54, -16.258, 78.572, 0, 27.685, 73.54]
  MoveL 390 to (76.64, -30.55, 1.69) mm, rotated rx -180 ry 0 rz 90 deg; joints [73.559, -16.205, 78.448, 0, 27.756, 73.559]
  MoveL 391 to (78.07, -30.03, 1.28) mm, rotated rx 180 ry 0 rz 90 deg; joints [73.588, -16.155, 78.337, 0, 27.818, 73.588]
  MoveL 392 to (79.36, -29.22, 0.87) mm, rotated rx -180 ry 0 rz 90 deg; joints [73.625, -16.111, 78.244, 0, 27.867, 73.625]
  MoveL 393 to (80.43, -28.14, 0.47) mm, rotated rx 180 ry 0 rz 90 deg; joints [73.668, -16.074, 78.173, 0, 27.901, 73.668]
  MoveL 394 to (81.23, -26.85, 0.06) mm, rotated rx 180 ry 0 rz 90 deg; joints [73.714, -16.044, 78.127, 0, 27.917, 73.714]
  MoveL 395 to (81.73, -25.41, -0.34) mm, rotated rx -180 ry 0 rz 90 deg; joints [73.763, -16.022, 78.107, 0, 27.915, 73.763]
  MoveL 396 to (81.87, -23.9, -0.75) mm, rotated rx 180 ry 0 rz 90 deg; joints [73.811, -16.009, 78.116, 0, 27.892, 73.811]
  MoveL 397 to (81.87, -5.21, -0.75) mm, rotated rx -180 ry 0 rz 90 deg; joints [74.388, -16.129, 78.522, 0, 27.607, 74.388]
  MoveL 398 to (81.84, -3.09, -0.75) mm, rotated rx -180 ry 0 rz 90 deg; joints [74.453, -16.143, 78.569, 0, 27.574, 74.453]
  MoveC 399 to (81.2, 1.25, -0.75) mm, rotated rx 180 ry 0 rz 90 deg; joints [74.583, -16.184, 78.709, 0, 27.475, 74.583] to (79.46, 5.28, -0.75) mm, rotated rx 180 ry 0 rz 90 deg; joints [74.693, -16.248, 78.925, 0, 27.323, 74.693]
  MoveC 400 to (74.36, 9.08, -0.75) mm, rotated rx -180 ry 0 rz 90 deg; joints [74.768, -16.384, 79.389, 0, 26.994, 74.768] to (68.07, 8.17, -0.75) mm, rotated rx -180 ry 0 rz 90 deg; joints [74.686, -16.515, 79.844, 0, 26.671, 74.686]
  MoveC 401 to (65, 5.91, -0.75) mm, rotated rx 180 ry 0 rz 90 deg; joints [74.589, -16.568, 80.028, 0, 26.54, 74.589] to (62.43, 3.1, -0.75) mm, rotated rx -180 ry 0 rz 90 deg; joints [74.478, -16.607, 80.162, 0, 26.445, 74.478]
  MoveL 402 to (60.48, 0.47, -0.75) mm, rotated rx -180 ry 0 rz 90 deg; joints [74.379, -16.633, 80.253, 0, 26.38, 74.379]
  MoveL 403 to (45.79, -19.71, -0.75) mm, rotated rx 180 ry 0 rz 90 deg; joints [73.614, -16.821, 80.914, 0, 25.907, 73.614]
  MoveC 404 to (43.74, -26.37, -0.75) mm, rotated rx -180 ry 0 rz 90 deg; joints [73.386, -16.823, 80.919, 0, 25.903, 73.386] to (46.21, -32.89, -0.75) mm, rotated rx -180 ry 0 rz 90 deg; joints [73.205, -16.73, 80.593, 0, 26.137, 73.205]
  MoveL 405 to (46.83, -33.64, -0.75) mm, rotated rx 180 ry 0 rz 90 deg; joints [73.187, -16.712, 80.53, 0, 26.182, 73.187]
  MoveL 406 to (63.02, -51.94, -0.75) mm, rotated rx 180 ry 0 rz 90 deg; joints [72.773, -16.242, 78.906, 0, 27.336, 72.773]
  MoveL 407 to (63.95, -52.91, -0.75) mm, rotated rx -180 ry 0 rz 90 deg; joints [72.752, -16.215, 78.813, 0, 27.402, 72.752]
  MoveC 408 to (67.85, -55.68, -0.75) mm, rotated rx -180 ry 0 rz 90 deg; joints [72.705, -16.109, 78.454, 0, 27.655, 72.705] to (72.49, -56.82, -0.75) mm, rotated rx -180 ry 0 rz 90 deg; joints [72.714, -15.997, 78.076, 0, 27.921, 72.714]
  MoveC 409 to (77.3, -55.13, -0.75) mm, rotated rx 180 ry 0 rz 90 deg; joints [72.811, -15.899, 77.751, 0, 28.149, 72.811] to (80.47, -51.14, -0.75) mm, rotated rx -180 ry 0 rz 90 deg; joints [72.963, -15.855, 77.603, 0, 28.252, 72.963]
  MoveC 410 to (81.44, -47.99, -0.75) mm, rotated rx 180 ry 0 rz 90 deg; joints [73.068, -15.855, 77.602, 0, 28.253, 73.068] to (81.83, -44.72, -0.75) mm, rotated rx 180 ry 0 rz 90 deg; joints [73.172, -15.869, 77.648, 0, 28.22, 73.172]
  MoveL 411 to (81.87, -43.12, -0.75) mm, rotated rx 180 ry 0 rz 90 deg; joints [73.221, -15.879, 77.682, 0, 28.197, 73.221]
  MoveL 412 to (81.87, -23.9, -0.75) mm, rotated rx 180 ry 0 rz 90 deg; joints [73.811, -16.009, 78.116, 0, 27.892, 73.811]
  MoveL 413 to (74.32, -23.9, -0.75) mm, rotated rx 180 ry 0 rz 90 deg; joints [73.743, -16.178, 78.69, 0, 27.489, 73.743]
  MoveL 414 to (74.32, -23.9, 2.25) mm, rotated rx -180 ry 0 rz 90 deg; joints [73.743, -16.329, 78.791, 0, 27.537, 73.743]
  Establecer velocidad (1000.0 mm/s)
  MoveL 415 to (74.32, -23.9, 10) mm, rotated rx -180 ry 0 rz 90 deg; joints [73.743, -16.716, 79.051, 0, 27.665, 73.743]
  Establecer velocidad (66.7 mm/s)
  MoveL 416 to (19.01, -75.15, 10) mm, rotated rx 180 ry 0 rz 90 deg; joints [71.616, -17.557, 81.961, 0, 25.596, 71.616]
  MoveL 417 to (19.01, -75.15, 2.5) mm, rotated rx 180 ry 0 rz 90 deg; joints [71.616, -17.179, 81.711, 0, 25.467, 71.616]
  MoveL 418 to (18.84, -76.66, 2.09) mm, rotated rx 180 ry 0 rz 90 deg; joints [71.567, -17.151, 81.674, 0, 25.478, 71.567]
  MoveL 419 to (19.04, -78.16, 1.69) mm, rotated rx -180 ry 0 rz 90 deg; joints [71.522, -17.117, 81.609, 0, 25.507, 71.522]
  MoveL 420 to (19.57, -79.59, 1.28) mm, rotated rx -180 ry 0 rz 90 deg; joints [71.483, -17.076, 81.523, 0, 25.553, 71.483]
  MoveL 421 to (20.4, -80.86, 0.87) mm, rotated rx -180 ry 0 rz 90 deg; joints [71.452, -17.03, 81.418, 0, 25.611, 71.452]
  MoveL 422 to (21.49, -81.92, 0.47) mm, rotated rx -180 ry 0 rz 90 deg; joints [71.431, -16.98, 81.3, 0, 25.68, 71.431]
  MoveL 423 to (22.78, -82.71, 0.06) mm, rotated rx 180 ry 0 rz 90 deg; joints [71.42, -16.927, 81.173, 0, 25.755, 71.42]
  MoveL 424 to (24.22, -83.2, -0.34) mm, rotated rx 180 ry 0 rz 90 deg; joints [71.42, -16.874, 81.042, 0, 25.832, 71.42]
  MoveL 425 to (25.74, -83.32, -0.75) mm, rotated rx -180 ry 0 rz 90 deg; joints [71.431, -16.822, 80.915, 0, 25.906, 71.431]
  MoveL 426 to (53.54, -83.04, -0.75) mm, rotated rx 180 ry 0 rz 90 deg; joints [71.725, -16.232, 78.87, 0, 27.362, 71.725]
  MoveL 427 to (55.96, -82.84, -0.75) mm, rotated rx -180 ry 0 rz 90 deg; joints [71.756, -16.18, 78.694, 0, 27.486, 71.756]
  MoveC 428 to (61.74, -80.52, -0.75) mm, rotated rx -180 ry 0 rz 90 deg; joints [71.885, -16.068, 78.317, 0, 27.751, 71.885] to (65.2, -75.34, -0.75) mm, rotated rx 180 ry 0 rz 90 deg; joints [72.077, -16.029, 78.183, 0, 27.845, 72.077]
  MoveC 429 to (65, -70.1, -0.75) mm, rotated rx 180 ry 0 rz 90 deg; joints [72.235, -16.071, 78.326, 0, 27.745, 72.235] to (62.66, -65.42, -0.75) mm, rotated rx -180 ry 0 rz 90 deg; joints [72.356, -16.156, 78.615, 0, 27.542, 72.356]
  MoveL 430 to (61.49, -63.97, -0.75) mm, rotated rx -180 ry 0 rz 90 deg; joints [72.389, -16.192, 78.737, 0, 27.455, 72.389]
  MoveL 431 to (34.48, -32.69, -0.75) mm, rotated rx -180 ry 0 rz 90 deg; joints [73.1, -16.975, 81.459, 0, 25.515, 73.1]
  MoveL 432 to (31.94, -29.85, -0.75) mm, rotated rx 180 ry 0 rz 90 deg; joints [73.165, -17.044, 81.708, 0, 25.336, 73.165]
  MoveL 433 to (31.75, -29.66, -0.75) mm, rotated rx -180 ry 0 rz 90 deg; joints [73.169, -17.049, 81.726, 0, 25.323, 73.169]
  MoveL 434 to (16.58, -17.49, -0.75) mm, rotated rx -180 ry 0 rz 90 deg; joints [73.41, -17.423, 83.089, 0, 24.334, 73.41]
  MoveL 435 to (14.85, -16.31, -0.75) mm, rotated rx -180 ry 0 rz 90 deg; joints [73.431, -17.463, 83.239, 0, 24.225, 73.431]
  MoveC 436 to (4.72, -15.08, -0.75) mm, rotated rx 180 ry 0 rz 90 deg; joints [73.374, -17.664, 83.989, 0, 23.674, 73.374] to (-2.14, -22.63, -0.75) mm, rotated rx 180 ry 0 rz 90 deg; joints [73.065, -17.75, 84.315, 0, 23.435, 73.065]
  MoveL 437 to (-14.44, -68.7, -0.75) mm, rotated rx 180 ry 0 rz 90 deg; joints [71.467, -17.704, 84.143, 0, 23.561, 71.467]
  MoveL 438 to (-14.71, -70.07, -0.75) mm, rotated rx 180 ry 0 rz 90 deg; joints [71.421, -17.701, 84.13, 0, 23.571, 71.421]
  MoveC 439 to (-12.62, -79.09, -0.75) mm, rotated rx 180 ry 0 rz 90 deg; joints [71.157, -17.605, 83.767, 0, 23.837, 71.157] to (-4.5, -83.52, -0.75) mm, rotated rx 180 ry 0 rz 90 deg; joints [71.105, -17.422, 83.085, 0, 24.337, 71.105]
  MoveL 440 to (-3.32, -83.61, -0.75) mm, rotated rx -180 ry 0 rz 90 deg; joints [71.115, -17.399, 82.999, 0, 24.399, 71.115]
  MoveL 441 to (25.74, -83.32, -0.75) mm, rotated rx -180 ry 0 rz 90 deg; joints [71.431, -16.822, 80.915, 0, 25.906, 71.431]
  MoveL 442 to (25.66, -75.77, -0.75) mm, rotated rx 180 ry 0 rz 90 deg; joints [71.665, -16.875, 81.104, 0, 25.771, 71.665]
  MoveL 443 to (25.66, -75.77, 2.25) mm, rotated rx 180 ry 0 rz 90 deg; joints [71.665, -17.026, 81.205, 0, 25.821, 71.665]
  Establecer velocidad (1000.0 mm/s)
  MoveL 444 to (25.66, -75.77, 10) mm, rotated rx -180 ry 0 rz 90 deg; joints [71.665, -17.417, 81.464, 0, 25.953, 71.665]
  Establecer velocidad (66.7 mm/s)
  MoveL 445 to (-76.09, -45.04, 10) mm, rotated rx 180 ry 0 rz 90 deg; joints [71.566, -19.448, 89.27, 0, 20.177, 71.566]
  MoveL 446 to (-76.09, -45.04, 2.5) mm, rotated rx 180 ry 0 rz 90 deg; joints [71.566, -19.057, 89.021, 0, 20.036, 71.566]
  MoveL 447 to (-77.59, -44.85, 2.09) mm, rotated rx 180 ry 0 rz 90 deg; joints [71.556, -19.06, 89.113, 0, 19.948, 71.556]
  MoveL 448 to (-79.1, -45.03, 1.69) mm, rotated rx 180 ry 0 rz 90 deg; joints [71.533, -19.061, 89.196, 0, 19.866, 71.533]
  MoveL 449 to (-80.53, -45.55, 1.28) mm, rotated rx 180 ry 0 rz 90 deg; joints [71.5, -19.06, 89.266, 0, 19.793, 71.5]
  MoveL 450 to (-81.82, -46.36, 0.87) mm, rotated rx -180 ry 0 rz 90 deg; joints [71.459, -19.054, 89.32, 0, 19.734, 71.459]
  MoveL 451 to (-82.89, -47.44, 0.47) mm, rotated rx 180 ry 0 rz 90 deg; joints [71.411, -19.043, 89.353, 0, 19.69, 71.411]
  MoveL 452 to (-83.69, -48.73, 0.06) mm, rotated rx 180 ry 0 rz 90 deg; joints [71.36, -19.028, 89.364, 0, 19.664, 71.36]
  MoveL 453 to (-84.19, -50.16, -0.34) mm, rotated rx 180 ry 0 rz 90 deg; joints [71.306, -19.007, 89.352, 0, 19.655, 71.306]
  MoveL 454 to (-84.33, -51.68, -0.75) mm, rotated rx 180 ry 0 rz 90 deg; joints [71.255, -18.98, 89.313, 0, 19.667, 71.255]
  MoveL 455 to (-84.33, -70.95, -0.75) mm, rotated rx 180 ry 0 rz 90 deg; joints [70.618, -18.878, 88.87, 0, 20.008, 70.618]
  MoveC 456 to (-80.62, -79.93, -0.75) mm, rotated rx 180 ry 0 rz 90 deg; joints [70.367, -18.771, 88.412, 0, 20.359, 70.367] to (-71.66, -83.68, -0.75) mm, rotated rx -180 ry 0 rz 90 deg; joints [70.349, -18.607, 87.722, 0, 20.885, 70.349]
  MoveL 457 to (-70.6, -83.69, -0.75) mm, rotated rx 180 ry 0 rz 90 deg; joints [70.361, -18.59, 87.65, 0, 20.94, 70.361]
  MoveL 458 to (-35.26, -83.41, -0.75) mm, rotated rx 180 ry 0 rz 90 deg; joints [70.772, -17.991, 85.245, 0, 22.746, 70.772]
  MoveC 459 to (-27.47, -80.7, -0.75) mm, rotated rx -180 ry 0 rz 90 deg; joints [70.944, -17.868, 84.769, 0, 23.099, 70.944] to (-22.93, -73.81, -0.75) mm, rotated rx 180 ry 0 rz 90 deg; joints [71.213, -17.829, 84.617, 0, 23.211, 71.213]
  MoveL 460 to (-10.23, -25.11, -0.75) mm, rotated rx 180 ry 0 rz 90 deg; joints [72.906, -17.885, 84.833, 0, 23.052, 72.906]
  MoveL 461 to (-10.04, -24.17, -0.75) mm, rotated rx -180 ry 0 rz 90 deg; joints [72.938, -17.887, 84.839, 0, 23.047, 72.938]
  MoveL 462 to (-9.95, -23.48, -0.75) mm, rotated rx 180 ry 0 rz 90 deg; joints [72.961, -17.889, 84.848, 0, 23.041, 72.961]
  MoveL 463 to (-9.91, -23.22, -0.75) mm, rotated rx 180 ry 0 rz 90 deg; joints [72.97, -17.89, 84.851, 0, 23.039, 72.97]
  MoveL 464 to (-9.82, -22.27, -0.75) mm, rotated rx 180 ry 0 rz 90 deg; joints [73.002, -17.893, 84.865, 0, 23.028, 73.002]
  MoveC 465 to (-11.3, -15.17, -0.75) mm, rotated rx -180 ry 0 rz 90 deg; joints [73.216, -17.959, 85.12, 0, 22.839, 73.216] to (-16.58, -10.21, -0.75) mm, rotated rx -180 ry 0 rz 90 deg; joints [73.326, -18.081, 85.596, 0, 22.485, 73.326]
  MoveC 466 to (-20.64, -9.14, -0.75) mm, rotated rx -180 ry 0 rz 90 deg; joints [73.321, -18.158, 85.901, 0, 22.257, 73.321] to (-24.83, -9.37, -0.75) mm, rotated rx 180 ry 0 rz 90 deg; joints [73.273, -18.231, 86.188, 0, 22.042, 73.273]
  MoveL 467 to (-74.18, -19.87, -0.75) mm, rotated rx -180 ry 0 rz 90 deg; joints [72.423, -18.984, 89.332, 0, 19.652, 72.423]
  MoveC 468 to (-81.47, -24.34, -0.75) mm, rotated rx -180 ry 0 rz 90 deg; joints [72.196, -19.073, 89.724, 0, 19.349, 72.196] to (-84.33, -32.4, -0.75) mm, rotated rx -180 ry 0 rz 90 deg; joints [71.896, -19.077, 89.74, 0, 19.337, 71.896]
  MoveL 469 to (-84.33, -51.68, -0.75) mm, rotated rx 180 ry 0 rz 90 deg; joints [71.255, -18.98, 89.313, 0, 19.667, 71.255]
  MoveL 470 to (-76.78, -51.68, -0.75) mm, rotated rx 180 ry 0 rz 90 deg; joints [71.339, -18.864, 88.81, 0, 20.054, 71.339]
  MoveL 471 to (-76.78, -51.68, 2.25) mm, rotated rx -180 ry 0 rz 90 deg; joints [71.339, -19.02, 88.91, 0, 20.11, 71.339]
  Establecer velocidad (1000.0 mm/s)
  MoveL 472 to (-76.78, -51.68, 10) mm, rotated rx 180 ry 0 rz 90 deg; joints [71.339, -19.423, 89.167, 0, 20.256, 71.339]
  Establecer velocidad (66.7 mm/s)
  MoveL 473 to (-76.09, 36.62, 10) mm, rotated rx 180 ry 0 rz 90 deg; joints [74.309, -19.829, 90.945, 0, 18.884, 74.309]
  MoveL 474 to (-76.09, 36.62, 2.5) mm, rotated rx 180 ry 0 rz 90 deg; joints [74.309, -19.436, 90.696, 0, 18.739, 74.309]
  MoveL 475 to (-77.59, 36.81, 2.09) mm, rotated rx 180 ry 0 rz 90 deg; joints [74.301, -19.437, 90.787, 0, 18.651, 74.301]
  MoveL 476 to (-79.1, 36.62, 1.69) mm, rotated rx -180 ry 0 rz 90 deg; joints [74.281, -19.437, 90.87, 0, 18.567, 74.281]
  MoveL 477 to (-80.53, 36.11, 1.28) mm, rotated rx -180 ry 0 rz 90 deg; joints [74.249, -19.434, 90.942, 0, 18.492, 74.249]
  MoveL 478 to (-81.82, 35.3, 0.87) mm, rotated rx 180 ry 0 rz 90 deg; joints [74.209, -19.428, 90.998, 0, 18.43, 74.209]
  MoveL 479 to (-82.89, 34.22, 0.47) mm, rotated rx 180 ry 0 rz 90 deg; joints [74.162, -19.418, 91.035, 0, 18.382, 74.162]
  MoveL 480 to (-83.69, 32.93, 0.06) mm, rotated rx 180 ry 0 rz 90 deg; joints [74.11, -19.403, 91.051, 0, 18.352, 74.11]
  MoveL 481 to (-84.19, 31.49, -0.34) mm, rotated rx -180 ry 0 rz 90 deg; joints [74.056, -19.382, 91.043, 0, 18.339, 74.056]
  MoveL 482 to (-84.33, 29.98, -0.75) mm, rotated rx -180 ry 0 rz 90 deg; joints [74.003, -19.357, 91.01, 0, 18.347, 74.003]
  MoveL 483 to (-84.32, 0.4, -0.75) mm, rotated rx 180 ry 0 rz 90 deg; joints [72.998, -19.23, 90.428, 0, 18.802, 72.998]
  MoveC 484 to (-79.74, -9.31, -0.75) mm, rotated rx 180 ry 0 rz 90 deg; joints [72.718, -19.118, 89.924, 0, 19.194, 72.718] to (-69.32, -11.94, -0.75) mm, rotated rx 180 ry 0 rz 90 deg; joints [72.739, -18.948, 89.174, 0, 19.774, 72.739]
  MoveL 485 to (-67.76, -11.63, -0.75) mm, rotated rx 180 ry 0 rz 90 deg; joints [72.765, -18.925, 89.075, 0, 19.851, 72.765]
  MoveL 486 to (-24.17, -1.59, -0.75) mm, rotated rx 180 ry 0 rz 90 deg; joints [73.533, -18.259, 86.303, 0, 21.956, 73.533]
  MoveL 487 to (-18.59, -0.31, -0.75) mm, rotated rx -180 ry 0 rz 90 deg; joints [73.629, -18.168, 85.941, 0, 22.227, 73.629]
  MoveC 488 to (-10.44, 5.8, -0.75) mm, rotated rx -180 ry 0 rz 90 deg; joints [73.905, -18.055, 85.495, 0, 22.56, 73.905] to (-9.51, 15.94, -0.75) mm, rotated rx -180 ry 0 rz 90 deg; joints [74.245, -18.09, 85.633, 0, 22.458, 74.245]
  MoveL 489 to (-9.73, 16.58, -0.75) mm, rotated rx 180 ry 0 rz 90 deg; joints [74.264, -18.098, 85.661, 0, 22.437, 74.264]
  MoveL 490 to (-16.47, 35.44, -0.75) mm, rotated rx -180 ry 0 rz 90 deg; joints [74.822, -18.308, 86.499, 0, 21.81, 74.822]
  MoveC 491 to (-18.54, 39.16, -0.75) mm, rotated rx 180 ry 0 rz 90 deg; joints [74.926, -18.361, 86.713, 0, 21.648, 74.926] to (-21.7, 42.01, -0.75) mm, rotated rx 180 ry 0 rz 90 deg; joints [74.992, -18.428, 86.986, 0, 21.443, 74.992]
  MoveL 492 to (-63.97, 69.14, -0.75) mm, rotated rx 180 ry 0 rz 90 deg; joints [75.531, -19.216, 90.363, 0, 18.853, 75.531]
  MoveL 493 to (-65.52, 70.01, -0.75) mm, rotated rx 180 ry 0 rz 90 deg; joints [75.547, -19.242, 90.482, 0, 18.76, 75.547]
  MoveC 494 to (-71.82, 71.72, -0.75) mm, rotated rx 180 ry 0 rz 90 deg; joints [75.55, -19.34, 90.934, 0, 18.407, 75.55] to (-78.18, 70.25, -0.75) mm, rotated rx 180 ry 0 rz 90 deg; joints [75.443, -19.426, 91.332, 0, 18.094, 75.443]
  MoveC 495 to (-82.62, 65.69, -0.75) mm, rotated rx 180 ry 0 rz 90 deg; joints [75.246, -19.472, 91.548, 0, 17.924, 75.246] to (-84.31, 59.57, -0.75) mm, rotated rx -180 ry 0 rz 90 deg; joints [75.019, -19.472, 91.552, 0, 17.92, 75.019]
  MoveL 496 to (-84.33, 58.28, -0.75) mm, rotated rx 180 ry 0 rz 90 deg; joints [74.974, -19.468, 91.531, 0, 17.937, 74.974]
  MoveL 497 to (-84.33, 29.98, -0.75) mm, rotated rx -180 ry 0 rz 90 deg; joints [74.003, -19.357, 91.01, 0, 18.347, 74.003]
  MoveL 498 to (-76.78, 29.98, -0.75) mm, rotated rx 180 ry 0 rz 90 deg; joints [74.077, -19.248, 90.508, 0, 18.74, 74.077]
  MoveL 499 to (-76.78, 29.98, 2.25) mm, rotated rx 180 ry 0 rz 90 deg; joints [74.077, -19.405, 90.609, 0, 18.797, 74.077]
  Establecer velocidad (1000.0 mm/s)
  MoveL 500 to (-76.78, 29.98, 10) mm, rotated rx -180 ry 0 rz 90 deg; joints [74.077, -19.812, 90.866, 0, 18.946, 74.077]
  Establecer velocidad (66.7 mm/s)
  MoveL 501 to (-75.33, 36.62, 10) mm, rotated rx -180 ry 0 rz 90 deg; joints [74.317, -19.818, 90.895, 0, 18.923, 74.317]
  MoveL 502 to (-75.33, 36.62, 2.25) mm, rotated rx 180 ry 0 rz 90 deg; joints [74.317, -19.411, 90.637, 0, 18.774, 74.317]
  MoveL 503 to (-76.83, 36.81, 1.84) mm, rotated rx 180 ry 0 rz 90 deg; joints [74.309, -19.413, 90.728, 0, 18.685, 74.309]
  MoveL 504 to (-78.34, 36.62, 1.44) mm, rotated rx -180 ry 0 rz 90 deg; joints [74.288, -19.413, 90.811, 0, 18.602, 74.288]
  MoveL 505 to (-79.77, 36.11, 1.03) mm, rotated rx 180 ry 0 rz 90 deg; joints [74.257, -19.41, 90.883, 0, 18.527, 74.257]
  MoveL 506 to (-81.05, 35.3, 0.62) mm, rotated rx -180 ry 0 rz 90 deg; joints [74.216, -19.404, 90.939, 0, 18.465, 74.216]
  MoveL 507 to (-82.12, 34.22, 0.22) mm, rotated rx 180 ry 0 rz 90 deg; joints [74.169, -19.394, 90.976, 0, 18.417, 74.169]
  MoveL 508 to (-82.93, 32.93, -0.19) mm, rotated rx 180 ry 0 rz 90 deg; joints [74.117, -19.378, 90.992, 0, 18.387, 74.117]
  MoveL 509 to (-83.43, 31.49, -0.59) mm, rotated rx 180 ry 0 rz 90 deg; joints [74.063, -19.358, 90.984, 0, 18.374, 74.063]
  MoveL 510 to (-83.57, 29.98, -1) mm, rotated rx -180 ry 0 rz 90 deg; joints [74.011, -19.333, 90.951, 0, 18.382, 74.011]
  MoveL 511 to (-83.56, 0.47, -1) mm, rotated rx 180 ry 0 rz 90 deg; joints [73.008, -19.206, 90.371, 0, 18.835, 73.008]
  MoveC 512 to (-79.35, -8.64, -1) mm, rotated rx -180 ry 0 rz 90 deg; joints [72.745, -19.103, 89.904, 0, 19.198, 72.745] to (-69.65, -11.22, -1) mm, rotated rx -180 ry 0 rz 90 deg; joints [72.759, -18.943, 89.202, 0, 19.741, 72.759]
  MoveL 513 to (-68.7, -11.05, -1) mm, rotated rx -180 ry 0 rz 90 deg; joints [72.775, -18.93, 89.142, 0, 19.788, 72.775]
  MoveL 514 to (-18.48, 0.52, -1) mm, rotated rx -180 ry 0 rz 90 deg; joints [73.657, -18.158, 85.942, 0, 22.216, 73.657]
  MoveC 515 to (-11.04, 6.27, -1) mm, rotated rx 180 ry 0 rz 90 deg; joints [73.915, -18.056, 85.538, 0, 22.517, 73.915] to (-10.21, 15.64, -1) mm, rotated rx -180 ry 0 rz 90 deg; joints [74.228, -18.088, 85.668, 0, 22.421, 74.228]
  MoveL 516 to (-10.53, 16.58, -1) mm, rotated rx 180 ry 0 rz 90 deg; joints [74.256, -18.099, 85.709, 0, 22.39, 74.256]
  MoveL 517 to (-17.18, 35.16, -1) mm, rotated rx -180 ry 0 rz 90 deg; joints [74.806, -18.306, 86.534, 0, 21.772, 74.806]
  MoveC 518 to (-19.14, 38.67, -1) mm, rotated rx 180 ry 0 rz 90 deg; joints [74.904, -18.356, 86.737, 0, 21.619, 74.904] to (-22.12, 41.37, -1) mm, rotated rx -180 ry 0 rz 90 deg; joints [74.967, -18.42, 86.995, 0, 21.425, 74.967]
  MoveL 519 to (-63.97, 68.23, -1) mm, rotated rx 180 ry 0 rz 90 deg; joints [75.5, -19.199, 90.338, 0, 18.861, 75.5]
  MoveL 520 to (-65.22, 68.99, -1) mm, rotated rx -180 ry 0 rz 90 deg; joints [75.515, -19.221, 90.436, 0, 18.785, 75.515]
  MoveC 521 to (-70.61, 70.84, -1) mm, rotated rx -180 ry 0 rz 90 deg; joints [75.531, -19.306, 90.829, 0, 18.477, 75.531] to (-76.29, 70.3, -1) mm, rotated rx 180 ry 0 rz 90 deg; joints [75.461, -19.386, 91.199, 0, 18.187, 75.461]
  MoveC 522 to (-81.5, 66.09, -1) mm, rotated rx 180 ry 0 rz 90 deg; joints [75.269, -19.444, 91.472, 0, 17.972, 75.269] to (-83.54, 59.71, -1) mm, rotated rx 180 ry 0 rz 90 deg; joints [75.031, -19.449, 91.495, 0, 17.954, 75.031]
  MoveL 523 to (-83.57, 58.28, -1) mm, rotated rx 180 ry 0 rz 90 deg; joints [74.981, -19.444, 91.472, 0, 17.972, 74.981]
  MoveL 524 to (-83.57, 29.98, -1) mm, rotated rx -180 ry 0 rz 90 deg; joints [74.011, -19.333, 90.951, 0, 18.382, 74.011]
  MoveL 525 to (-76.02, 29.98, -1) mm, rotated rx -180 ry 0 rz 90 deg; joints [74.084, -19.223, 90.449, 0, 18.774, 74.084]
  MoveL 526 to (-76.02, 29.98, 2) mm, rotated rx 180 ry 0 rz 90 deg; joints [74.084, -19.381, 90.549, 0, 18.831, 74.084]
  Establecer velocidad (1000.0 mm/s)
  MoveL 527 to (-76.02, 29.98, 10) mm, rotated rx 180 ry 0 rz 90 deg; joints [74.084, -19.8, 90.815, 0, 18.985, 74.084]
  Establecer velocidad (66.7 mm/s)
  MoveL 528 to (-75.33, -45.03, 10) mm, rotated rx 180 ry 0 rz 90 deg; joints [71.575, -19.436, 89.219, 0, 20.216, 71.575]
  MoveL 529 to (-75.33, -45.03, 2.25) mm, rotated rx -180 ry 0 rz 90 deg; joints [71.575, -19.032, 88.962, 0, 20.07, 71.575]
  MoveL 530 to (-76.83, -44.85, 1.84) mm, rotated rx -180 ry 0 rz 90 deg; joints [71.564, -19.036, 89.054, 0, 19.982, 71.564]
  MoveL 531 to (-78.34, -45.03, 1.44) mm, rotated rx -180 ry 0 rz 90 deg; joints [71.542, -19.037, 89.137, 0, 19.9, 71.542]
  MoveL 532 to (-79.77, -45.54, 1.03) mm, rotated rx -180 ry 0 rz 90 deg; joints [71.509, -19.035, 89.207, 0, 19.828, 71.509]
  MoveL 533 to (-81.05, -46.36, 0.62) mm, rotated rx 180 ry 0 rz 90 deg; joints [71.468, -19.029, 89.261, 0, 19.768, 71.468]
  MoveL 534 to (-82.12, -47.43, 0.22) mm, rotated rx 180 ry 0 rz 90 deg; joints [71.42, -19.019, 89.294, 0, 19.724, 71.42]
  MoveL 535 to (-82.93, -48.72, -0.19) mm, rotated rx 180 ry 0 rz 90 deg; joints [71.368, -19.003, 89.305, 0, 19.698, 71.368]
  MoveL 536 to (-83.43, -50.16, -0.59) mm, rotated rx -180 ry 0 rz 90 deg; joints [71.315, -18.982, 89.293, 0, 19.689, 71.315]
  MoveL 537 to (-83.57, -51.67, -1) mm, rotated rx -180 ry 0 rz 90 deg; joints [71.263, -18.955, 89.254, 0, 19.701, 71.263]
  MoveL 538 to (-83.57, -70.94, -1) mm, rotated rx 180 ry 0 rz 90 deg; joints [70.628, -18.853, 88.812, 0, 20.042, 70.628]
  MoveC 539 to (-80.09, -79.38, -1) mm, rotated rx 180 ry 0 rz 90 deg; joints [70.391, -18.753, 88.38, 0, 20.372, 70.391] to (-71.66, -82.91, -1) mm, rotated rx 180 ry 0 rz 90 deg; joints [70.374, -18.598, 87.731, 0, 20.867, 70.374]
  MoveL 540 to (-70.6, -82.92, -1) mm, rotated rx 180 ry 0 rz 90 deg; joints [70.386, -18.581, 87.66, 0, 20.921, 70.386]
  MoveL 541 to (-35.54, -82.65, -1) mm, rotated rx 180 ry 0 rz 90 deg; joints [70.793, -17.988, 85.274, 0, 22.714, 70.793]
  MoveC 542 to (-27.97, -80.11, -1) mm, rotated rx -180 ry 0 rz 90 deg; joints [70.958, -17.868, 84.81, 0, 23.058, 70.958] to (-23.59, -73.44, -1) mm, rotated rx -180 ry 0 rz 90 deg; joints [71.218, -17.83, 84.664, 0, 23.167, 71.218]
  MoveL 543 to (-11.03, -25.11, -1) mm, rotated rx 180 ry 0 rz 90 deg; joints [72.898, -17.886, 84.88, 0, 23.006, 72.898]
  MoveL 544 to (-10.74, -23.75, -1) mm, rotated rx 180 ry 0 rz 90 deg; joints [72.945, -17.889, 84.889, 0, 23, 72.945]
  MoveC 545 to (-11.33, -16.92, -1) mm, rotated rx -180 ry 0 rz 90 deg; joints [73.159, -17.937, 85.077, 0, 22.86, 73.159] to (-15.64, -11.6, -1) mm, rotated rx -180 ry 0 rz 90 deg; joints [73.29, -18.044, 85.492, 0, 22.552, 73.29]
  MoveC 546 to (-19.76, -10.03, -1) mm, rotated rx -180 ry 0 rz 90 deg; joints [73.301, -18.125, 85.813, 0, 22.313, 73.301] to (-24.17, -10.04, -1) mm, rotated rx 180 ry 0 rz 90 deg; joints [73.257, -18.203, 86.12, 0, 22.083, 73.257]
  MoveL 547 to (-25.11, -10.22, -1) mm, rotated rx 180 ry 0 rz 90 deg; joints [73.242, -18.218, 86.182, 0, 22.037, 73.242]
  MoveL 548 to (-74.03, -20.62, -1) mm, rotated rx -180 ry 0 rz 90 deg; joints [72.4, -18.965, 89.298, 0, 19.668, 72.4]
  MoveC 549 to (-80.88, -24.83, -1) mm, rotated rx -180 ry 0 rz 90 deg; joints [72.186, -19.049, 89.666, 0, 19.383, 72.186] to (-83.57, -32.4, -1) mm, rotated rx -180 ry 0 rz 90 deg; joints [71.904, -19.052, 89.681, 0, 19.371, 71.904]
  MoveL 550 to (-83.57, -51.67, -1) mm, rotated rx -180 ry 0 rz 90 deg; joints [71.263, -18.955, 89.254, 0, 19.701, 71.263]
  MoveL 551 to (-76.02, -51.67, -1) mm, rotated rx -180 ry 0 rz 90 deg; joints [71.348, -18.839, 88.751, 0, 20.089, 71.348]
  MoveL 552 to (-76.02, -51.67, 2) mm, rotated rx -180 ry 0 rz 90 deg; joints [71.348, -18.995, 88.851, 0, 20.144, 71.348]
  Establecer velocidad (1000.0 mm/s)
  MoveL 553 to (-76.02, -51.67, 10) mm, rotated rx 180 ry 0 rz 90 deg; joints [71.348, -19.412, 89.117, 0, 20.295, 71.348]
  Establecer velocidad (66.7 mm/s)
  MoveL 554 to (18.88, -74.41, 10) mm, rotated rx 180 ry 0 rz 90 deg; joints [71.638, -17.565, 81.989, 0, 25.576, 71.638]
  MoveL 555 to (18.88, -74.41, 2.25) mm, rotated rx 180 ry 0 rz 90 deg; joints [71.638, -17.174, 81.73, 0, 25.443, 71.638]
  MoveL 556 to (18.71, -75.91, 1.84) mm, rotated rx 180 ry 0 rz 90 deg; joints [71.589, -17.147, 81.693, 0, 25.454, 71.589]
  MoveL 557 to (18.91, -77.42, 1.44) mm, rotated rx -180 ry 0 rz 90 deg; joints [71.544, -17.112, 81.628, 0, 25.483, 71.544]
  MoveL 558 to (19.44, -78.85, 1.03) mm, rotated rx 180 ry 0 rz 90 deg; joints [71.505, -17.071, 81.542, 0, 25.529, 71.505]
  MoveL 559 to (20.26, -80.12, 0.62) mm, rotated rx 180 ry 0 rz 90 deg; joints [71.474, -17.025, 81.438, 0, 25.587, 71.474]
  MoveL 560 to (21.35, -81.18, 0.22) mm, rotated rx -180 ry 0 rz 90 deg; joints [71.452, -16.975, 81.319, 0, 25.656, 71.452]
  MoveL 561 to (22.65, -81.97, -0.19) mm, rotated rx 180 ry 0 rz 90 deg; joints [71.441, -16.923, 81.192, 0, 25.731, 71.441]
  MoveL 562 to (24.09, -82.45, -0.59) mm, rotated rx -180 ry 0 rz 90 deg; joints [71.441, -16.869, 81.062, 0, 25.808, 71.441]
  MoveL 563 to (25.6, -82.58, -1) mm, rotated rx -180 ry 0 rz 90 deg; joints [71.453, -16.817, 80.935, 0, 25.882, 71.453]
  MoveL 564 to (52.59, -82.3, -1) mm, rotated rx 180 ry 0 rz 90 deg; joints [71.738, -16.245, 78.951, 0, 27.295, 71.738]
  MoveL 565 to (54.98, -82.2, -1) mm, rotated rx -180 ry 0 rz 90 deg; joints [71.766, -16.193, 78.774, 0, 27.419, 71.766]
  MoveC 566 to (59.93, -80.77, -1) mm, rotated rx 180 ry 0 rz 90 deg; joints [71.859, -16.094, 78.439, 0, 27.655, 71.859] to (63.66, -77.23, -1) mm, rotated rx -180 ry 0 rz 90 deg; joints [72.004, -16.037, 78.245, 0, 27.792, 72.004]
  MoveC 567 to (64.59, -71.88, -1) mm, rotated rx -180 ry 0 rz 90 deg; joints [72.177, -16.055, 78.305, 0, 27.75, 72.177] to (62.65, -66.81, -1) mm, rotated rx 180 ry 0 rz 90 deg; joints [72.313, -16.134, 78.574, 0, 27.561, 72.313]
  MoveL 568 to (61.29, -64.91, -1) mm, rotated rx -180 ry 0 rz 90 deg; joints [72.358, -16.178, 78.721, 0, 27.457, 72.358]
  MoveL 569 to (53.54, -55.91, -1) mm, rotated rx 180 ry 0 rz 90 deg; joints [72.56, -16.41, 79.514, 0, 26.896, 72.56]
  MoveL 570 to (53.14, -55.44, -1) mm, rotated rx -180 ry 0 rz 90 deg; joints [72.57, -16.422, 79.555, 0, 26.866, 72.57]
  MoveL 571 to (34.28, -33.64, -1) mm, rotated rx -180 ry 0 rz 90 deg; joints [73.068, -16.96, 81.444, 0, 25.516, 73.068]
  MoveL 572 to (31.75, -30.75, -1) mm, rotated rx -180 ry 0 rz 90 deg; joints [73.135, -17.03, 81.693, 0, 25.336, 73.135]
  MoveL 573 to (30.8, -29.84, -1) mm, rotated rx -180 ry 0 rz 90 deg; joints [73.154, -17.054, 81.783, 0, 25.272, 73.154]
  MoveL 574 to (15.64, -17.74, -1) mm, rotated rx 180 ry 0 rz 90 deg; joints [73.393, -17.427, 83.143, 0, 24.284, 73.393]
  MoveL 575 to (14.69, -17.09, -1) mm, rotated rx 180 ry 0 rz 90 deg; joints [73.405, -17.449, 83.225, 0, 24.224, 73.405]
  MoveC 576 to (9.61, -15.24, -1) mm, rotated rx 180 ry 0 rz 90 deg; joints [73.416, -17.557, 83.628, 0, 23.929, 73.416] to (4.26, -16.02, -1) mm, rotated rx 180 ry 0 rz 90 deg; joints [73.34, -17.654, 83.993, 0, 23.661, 73.34]
  MoveC 577 to (0.59, -19, -1) mm, rotated rx -180 ry 0 rz 90 deg; joints [73.209, -17.706, 84.191, 0, 23.515, 73.209] to (-1.54, -23.22, -1) mm, rotated rx 180 ry 0 rz 90 deg; joints [73.052, -17.722, 84.251, 0, 23.471, 73.052]
  MoveL 578 to (-13.8, -69.43, -1) mm, rotated rx 180 ry 0 rz 90 deg; joints [71.451, -17.675, 84.073, 0, 23.602, 71.451]
  MoveC 579 to (-12.03, -78.55, -1) mm, rotated rx 180 ry 0 rz 90 deg; joints [71.181, -17.584, 83.731, 0, 23.854, 71.181] to (-3.77, -82.82, -1) mm, rotated rx -180 ry 0 rz 90 deg; joints [71.135, -17.4, 83.043, 0, 24.357, 71.135]
  MoveL 580 to (-2.37, -82.86, -1) mm, rotated rx 180 ry 0 rz 90 deg; joints [71.149, -17.373, 82.942, 0, 24.431, 71.149]
  MoveL 581 to (25.6, -82.58, -1) mm, rotated rx -180 ry 0 rz 90 deg; joints [71.453, -16.817, 80.935, 0, 25.882, 71.453]
  MoveL 582 to (25.53, -75.03, -1) mm, rotated rx 180 ry 0 rz 90 deg; joints [71.687, -16.87, 81.124, 0, 25.746, 71.687]
  MoveL 583 to (25.53, -75.03, 2) mm, rotated rx 180 ry 0 rz 90 deg; joints [71.687, -17.021, 81.225, 0, 25.797, 71.687]
  Establecer velocidad (1000.0 mm/s)
  MoveL 584 to (25.53, -75.03, 10) mm, rotated rx 180 ry 0 rz 90 deg; joints [71.687, -17.425, 81.492, 0, 25.933, 71.687]
  Establecer velocidad (66.7 mm/s)
  MoveL 585 to (72.86, -30.55, 10) mm, rotated rx 180 ry 0 rz 90 deg; joints [73.525, -16.705, 79.014, 0, 27.691, 73.525]
  MoveL 586 to (72.86, -30.55, 2.25) mm, rotated rx 180 ry 0 rz 90 deg; joints [73.525, -16.318, 78.754, 0, 27.564, 73.525]
  MoveL 587 to (74.37, -30.73, 1.84) mm, rotated rx -180 ry 0 rz 90 deg; joints [73.533, -16.262, 78.622, 0, 27.64, 73.533]
  MoveL 588 to (75.88, -30.55, 1.44) mm, rotated rx -180 ry 0 rz 90 deg; joints [73.552, -16.209, 78.498, 0, 27.711, 73.552]
  MoveL 589 to (77.31, -30.04, 1.03) mm, rotated rx -180 ry 0 rz 90 deg; joints [73.581, -16.16, 78.387, 0, 27.773, 73.581]
  MoveL 590 to (78.59, -29.22, 0.62) mm, rotated rx 180 ry 0 rz 90 deg; joints [73.618, -16.116, 78.294, 0, 27.822, 73.618]
  MoveL 591 to (79.66, -28.14, 0.22) mm, rotated rx -180 ry 0 rz 90 deg; joints [73.661, -16.079, 78.223, 0, 27.856, 73.661]
  MoveL 592 to (80.46, -26.85, -0.19) mm, rotated rx 180 ry 0 rz 90 deg; joints [73.707, -16.049, 78.177, 0, 27.872, 73.707]
  MoveL 593 to (80.96, -25.42, -0.59) mm, rotated rx 180 ry 0 rz 90 deg; joints [73.756, -16.027, 78.157, 0, 27.87, 73.756]
  MoveL 594 to (81.1, -23.91, -1) mm, rotated rx -180 ry 0 rz 90 deg; joints [73.804, -16.013, 78.166, 0, 27.847, 73.804]
  MoveL 595 to (81.1, -5.21, -1) mm, rotated rx 180 ry 0 rz 90 deg; joints [74.381, -16.134, 78.572, 0, 27.562, 74.381]
  MoveL 596 to (81.06, -3.02, -1) mm, rotated rx -180 ry 0 rz 90 deg; joints [74.449, -16.148, 78.621, 0, 27.527, 74.449]
  MoveC 597 to (80.5, 0.91, -1) mm, rotated rx 180 ry 0 rz 90 deg; joints [74.566, -16.185, 78.747, 0, 27.439, 74.566] to (78.99, 4.59, -1) mm, rotated rx -180 ry 0 rz 90 deg; joints [74.667, -16.241, 78.938, 0, 27.304, 74.667]
  MoveC 598 to (74.05, 8.33, -1) mm, rotated rx 180 ry 0 rz 90 deg; joints [74.742, -16.373, 79.389, 0, 26.984, 74.742] to (67.95, 7.23, -1) mm, rotated rx 180 ry 0 rz 90 deg; joints [74.655, -16.5, 79.826, 0, 26.674, 74.655]
  MoveC 599 to (65.04, 4.89, -1) mm, rotated rx 180 ry 0 rz 90 deg; joints [74.557, -16.549, 79.996, 0, 26.553, 74.557] to (62.58, 2.07, -1) mm, rotated rx -180 ry 0 rz 90 deg; joints [74.447, -16.585, 80.121, 0, 26.464, 74.447]
  MoveL 600 to (46.91, -19.43, -1) mm, rotated rx 180 ry 0 rz 90 deg; joints [73.633, -16.787, 80.828, 0, 25.958, 73.633]
  MoveL 601 to (46.25, -20.37, -1) mm, rotated rx -180 ry 0 rz 90 deg; joints [73.597, -16.795, 80.857, 0, 25.938, 73.597]
  MoveC 602 to (44.51, -26.59, -1) mm, rotated rx -180 ry 0 rz 90 deg; joints [73.386, -16.792, 80.849, 0, 25.944, 73.386] to (46.91, -32.58, -1) mm, rotated rx -180 ry 0 rz 90 deg; joints [73.221, -16.705, 80.539, 0, 26.165, 73.221]
  MoveL 603 to (63.02, -50.8, -1) mm, rotated rx 180 ry 0 rz 90 deg; joints [72.808, -16.237, 78.924, 0, 27.313, 72.808]
  MoveL 604 to (64.23, -52.09, -1) mm, rotated rx -180 ry 0 rz 90 deg; joints [72.78, -16.202, 78.803, 0, 27.399, 72.78]
  MoveC 605 to (66.79, -54.21, -1) mm, rotated rx -180 ry 0 rz 90 deg; joints [72.74, -16.13, 78.561, 0, 27.57, 72.74] to (69.8, -55.62, -1) mm, rotated rx 180 ry 0 rz 90 deg; joints [72.725, -16.053, 78.3, 0, 27.753, 72.725]
  MoveC 606 to (75.49, -55.33, -1) mm, rotated rx 180 ry 0 rz 90 deg; joints [72.788, -15.927, 77.875, 0, 28.051, 72.788] to (79.54, -51.32, -1) mm, rotated rx 180 ry 0 rz 90 deg; joints [72.949, -15.863, 77.661, 0, 28.201, 72.949]
  MoveC 607 to (80.61, -48.13, -1) mm, rotated rx 180 ry 0 rz 90 deg; joints [73.056, -15.86, 77.653, 0, 28.207, 73.056] to (81.05, -44.79, -1) mm, rotated rx 180 ry 0 rz 90 deg; joints [73.162, -15.873, 77.698, 0, 28.176, 73.162]
  MoveL 608 to (81.1, -43.12, -1) mm, rotated rx 180 ry 0 rz 90 deg; joints [73.214, -15.884, 77.732, 0, 28.152, 73.214]
  MoveL 609 to (81.1, -23.91, -1) mm, rotated rx -180 ry 0 rz 90 deg; joints [73.804, -16.013, 78.166, 0, 27.847, 73.804]
  MoveL 610 to (73.55, -23.91, -1) mm, rotated rx 180 ry 0 rz 90 deg; joints [73.736, -16.183, 78.739, 0, 27.444, 73.736]
  MoveL 611 to (73.55, -23.91, 2) mm, rotated rx -180 ry 0 rz 90 deg; joints [73.736, -16.333, 78.841, 0, 27.492, 73.736]
  Establecer velocidad (1000.0 mm/s)
  MoveL 612 to (73.55, -23.91, 10) mm, rotated rx -180 ry 0 rz 90 deg; joints [73.736, -16.733, 79.109, 0, 27.624, 73.736]
  Establecer velocidad (66.7 mm/s)
  MoveL 613 to (38.15, 30.17, 10) mm, rotated rx -180 ry 0 rz 90 deg; joints [75.126, -17.807, 82.857, 0, 24.95, 75.126]
  MoveL 614 to (38.15, 30.17, 2.25) mm, rotated rx 180 ry 0 rz 90 deg; joints [75.126, -17.414, 82.599, 0, 24.815, 75.126]
  MoveL 615 to (38.29, 31.68, 1.84) mm, rotated rx -180 ry 0 rz 90 deg; joints [75.176, -17.399, 82.605, 0, 24.794, 75.176]
  MoveL 616 to (38.07, 33.18, 1.44) mm, rotated rx -180 ry 0 rz 90 deg; joints [75.222, -17.391, 82.636, 0, 24.754, 75.222]
  MoveL 617 to (37.52, 34.59, 1.03) mm, rotated rx 180 ry 0 rz 90 deg; joints [75.263, -17.389, 82.69, 0, 24.698, 75.263]
  MoveL 618 to (36.66, 35.85, 0.62) mm, rotated rx -180 ry 0 rz 90 deg; joints [75.296, -17.392, 82.763, 0, 24.629, 75.296]
  MoveL 619 to (35.56, 36.89, 0.22) mm, rotated rx 180 ry 0 rz 90 deg; joints [75.32, -17.398, 82.85, 0, 24.549, 75.32]
  MoveL 620 to (34.25, 37.66, -0.19) mm, rotated rx 180 ry 0 rz 90 deg; joints [75.334, -17.408, 82.946, 0, 24.462, 75.334]
  MoveL 621 to (32.8, 38.12, -0.59) mm, rotated rx 180 ry 0 rz 90 deg; joints [75.336, -17.418, 83.046, 0, 24.372, 75.336]
  MoveL 622 to (31.29, 38.22, -1) mm, rotated rx 180 ry 0 rz 90 deg; joints [75.327, -17.427, 83.144, 0, 24.283, 75.327]
  MoveL 623 to (7.11, 37.56, -1) mm, rotated rx 180 ry 0 rz 90 deg; joints [75.099, -17.883, 84.869, 0, 23.015, 75.099]
  MoveL 624 to (6.16, 37.44, -1) mm, rotated rx -180 ry 0 rz 90 deg; joints [75.087, -17.9, 84.934, 0, 22.967, 75.087]
  MoveL 625 to (5.21, 37.26, -1) mm, rotated rx 180 ry 0 rz 90 deg; joints [75.073, -17.917, 84.998, 0, 22.919, 75.073]
  MoveC 626 to (-1.77, 32.53, -1) mm, rotated rx 180 ry 0 rz 90 deg; joints [74.857, -18.021, 85.402, 0, 22.619, 74.857] to (-2.81, 24.17, -1) mm, rotated rx -180 ry 0 rz 90 deg; joints [74.574, -17.998, 85.314, 0, 22.684, 74.574]
  MoveL 627 to (-2.53, 23.22, -1) mm, rotated rx 180 ry 0 rz 90 deg; joints [74.546, -17.989, 85.276, 0, 22.713, 74.546]
  MoveL 628 to (2.96, 8.05, -1) mm, rotated rx 180 ry 0 rz 90 deg; joints [74.103, -17.81, 84.586, 0, 23.224, 74.103]
  MoveL 629 to (3.81, 5.85, -1) mm, rotated rx 180 ry 0 rz 90 deg; joints [74.04, -17.782, 84.481, 0, 23.302, 74.04]
  MoveC 630 to (5.16, 3.37, -1) mm, rotated rx -180 ry 0 rz 90 deg; joints [73.972, -17.744, 84.334, 0, 23.41, 73.972] to (7.13, 1.36, -1) mm, rotated rx 180 ry 0 rz 90 deg; joints [73.926, -17.696, 84.153, 0, 23.544, 73.926]
  MoveL 631 to (24.61, -12.25, -1) mm, rotated rx 180 ry 0 rz 90 deg; joints [73.653, -17.283, 82.613, 0, 24.67, 73.653]
  MoveC 632 to (32.17, -14.4, -1) mm, rotated rx 180 ry 0 rz 90 deg; joints [73.655, -17.12, 82.018, 0, 25.102, 73.655] to (39.1, -10.68, -1) mm, rotated rx 180 ry 0 rz 90 deg; joints [73.836, -17.001, 81.591, 0, 25.41, 73.836]
  MoveL 633 to (39.71, -9.95, -1) mm, rotated rx -180 ry 0 rz 90 deg; joints [73.865, -16.993, 81.561, 0, 25.431, 73.865]
  MoveL 634 to (62.17, 21.32, -1) mm, rotated rx 180 ry 0 rz 90 deg; joints [75.049, -16.706, 80.544, 0, 26.162, 75.049]
  MoveL 635 to (63.18, 22.82, -1) mm, rotated rx 180 ry 0 rz 90 deg; joints [75.104, -16.693, 80.498, 0, 26.195, 75.104]
  MoveC 636 to (64.93, 26.63, -1) mm, rotated rx -180 ry 0 rz 90 deg; joints [75.239, -16.677, 80.443, 0, 26.234, 75.239] to (65.34, 30.8, -1) mm, rotated rx -180 ry 0 rz 90 deg; joints [75.374, -16.692, 80.494, 0, 26.198, 75.374]
  MoveC 637 to (62.65, 36.01, -1) mm, rotated rx 180 ry 0 rz 90 deg; joints [75.517, -16.777, 80.796, 0, 25.982, 75.517] to (57.37, 38.57, -1) mm, rotated rx 180 ry 0 rz 90 deg; joints [75.554, -16.902, 81.237, 0, 25.665, 75.554]
  MoveC 638 to (55.01, 38.78, -1) mm, rotated rx -180 ry 0 rz 90 deg; joints [75.542, -16.952, 81.417, 0, 25.536, 75.542] to (52.63, 38.81, -1) mm, rotated rx -180 ry 0 rz 90 deg; joints [75.523, -17.002, 81.593, 0, 25.409, 75.523]
  MoveL 639 to (31.29, 38.22, -1) mm, rotated rx 180 ry 0 rz 90 deg; joints [75.327, -17.427, 83.144, 0, 24.283, 75.327]
  MoveL 640 to (31.49, 30.67, -1) mm, rotated rx 180 ry 0 rz 90 deg; joints [75.086, -17.384, 82.985, 0, 24.399, 75.086]
  MoveL 641 to (31.49, 30.67, 2) mm, rotated rx 180 ry 0 rz 90 deg; joints [75.086, -17.537, 83.085, 0, 24.451, 75.086]
  Establecer velocidad (1000.0 mm/s)
  MoveL 642 to (31.49, 30.67, 10) mm, rotated rx -180 ry 0 rz 90 deg; joints [75.086, -17.943, 83.352, 0, 24.591, 75.086]
  Establecer velocidad (66.7 mm/s)
  MoveL 643 to (26.56, 74.14, 10) mm, rotated rx 180 ry 0 rz 90 deg; joints [76.452, -18.254, 84.506, 0, 23.748, 76.452]
  MoveL 644 to (26.56, 74.14, 2.25) mm, rotated rx -180 ry 0 rz 90 deg; joints [76.452, -17.859, 84.249, 0, 23.61, 76.452]
  MoveL 645 to (26.76, 75.64, 1.84) mm, rotated rx 180 ry 0 rz 90 deg; joints [76.503, -17.841, 84.246, 0, 23.595, 76.503]
  MoveL 646 to (26.6, 77.16, 1.44) mm, rotated rx -180 ry 0 rz 90 deg; joints [76.551, -17.83, 84.27, 0, 23.56, 76.551]
  MoveL 647 to (26.11, 78.59, 1.03) mm, rotated rx 180 ry 0 rz 90 deg; joints [76.594, -17.825, 84.317, 0, 23.508, 76.594]
  MoveL 648 to (25.31, 79.89, 0.62) mm, rotated rx -180 ry 0 rz 90 deg; joints [76.63, -17.826, 84.383, 0, 23.443, 76.63]
  MoveL 649 to (24.25, 80.97, 0.22) mm, rotated rx 180 ry 0 rz 90 deg; joints [76.657, -17.83, 84.465, 0, 23.365, 76.657]
  MoveL 650 to (22.97, 81.79, -0.19) mm, rotated rx 180 ry 0 rz 90 deg; joints [76.674, -17.837, 84.557, 0, 23.28, 76.674]
  MoveL 651 to (21.54, 82.31, -0.59) mm, rotated rx 180 ry 0 rz 90 deg; joints [76.68, -17.845, 84.655, 0, 23.19, 76.68]
  MoveL 652 to (20.03, 82.47, -1) mm, rotated rx -180 ry 0 rz 90 deg; joints [76.673, -17.853, 84.752, 0, 23.101, 76.673]
  MoveC 653 to (-5.73, 82.77, -1) mm, rotated rx 180 ry 0 rz 90 deg; joints [76.48, -18.319, 86.585, 0, 21.734, 76.48] to (-31.49, 82.96, -1) mm, rotated rx 180 ry 0 rz 90 deg; joints [76.278, -18.752, 88.38, 0, 20.372, 76.278]
  MoveC 654 to (-36.46, 82.38, -1) mm, rotated rx -180 ry 0 rz 90 deg; joints [76.217, -18.83, 88.712, 0, 20.118, 76.217] to (-41.15, 80.61, -1) mm, rotated rx 180 ry 0 rz 90 deg; joints [76.118, -18.898, 89.004, 0, 19.894, 76.118]
  MoveC 655 to (-45.29, 75.33, -1) mm, rotated rx -180 ry 0 rz 90 deg; joints [75.904, -18.942, 89.196, 0, 19.746, 75.904] to (-44.06, 68.74, -1) mm, rotated rx -180 ry 0 rz 90 deg; joints [75.691, -18.897, 88.999, 0, 19.898, 75.691]
  MoveC 656 to (-41.29, 65.51, -1) mm, rotated rx -180 ry 0 rz 90 deg; joints [75.606, -18.84, 88.753, 0, 20.087, 75.606] to (-37.94, 62.89, -1) mm, rotated rx 180 ry 0 rz 90 deg; joints [75.547, -18.775, 88.477, 0, 20.298, 75.547]
  MoveL 657 to (-14.95, 48.35, -1) mm, rotated rx 180 ry 0 rz 90 deg; joints [75.261, -18.328, 86.624, 0, 21.704, 75.261]
  MoveC 658 to (-10.88, 46.6, -1) mm, rotated rx 180 ry 0 rz 90 deg; joints [75.239, -18.25, 86.308, 0, 21.942, 75.239] to (-6.47, 46.22, -1) mm, rotated rx 180 ry 0 rz 90 deg; joints [75.265, -18.17, 85.991, 0, 22.179, 75.265]
  MoveL 659 to (68.74, 51.65, -1) mm, rotated rx 180 ry 0 rz 90 deg; joints [76.061, -16.732, 80.636, 0, 26.096, 76.061]
  MoveL 660 to (72.14, 51.86, -1) mm, rotated rx 180 ry 0 rz 90 deg; joints [76.094, -16.661, 80.386, 0, 26.275, 76.094]
  MoveC 661 to (78.21, 54.73, -1) mm, rotated rx -180 ry 0 rz 90 deg; joints [76.232, -16.545, 79.982, 0, 26.563, 76.232] to (80.68, 60.97, -1) mm, rotated rx -180 ry 0 rz 90 deg; joints [76.448, -16.524, 79.91, 0, 26.614, 76.448]
  MoveL 662 to (80.67, 72.49, -1) mm, rotated rx 180 ry 0 rz 90 deg; joints [76.812, -16.584, 80.117, 0, 26.467, 76.812]
  MoveC 663 to (77.97, 78.9, -1) mm, rotated rx 180 ry 0 rz 90 deg; joints [76.995, -16.674, 80.434, 0, 26.241, 76.995] to (71.55, 81.55, -1) mm, rotated rx -180 ry 0 rz 90 deg; joints [77.032, -16.824, 80.962, 0, 25.863, 77.032]
